LIN {X 0,Y 530.663,Z 618.387,A -85,B 0,C 180,E1 -4307.378,E2 -4307.378} C_VEL
LIN {X 0,Y 530.971,Z 618.347,A -85,B 0,C 180,E1 -4309.321,E2 -4309.321} C_VEL
LIN {X 0,Y 531.057,Z 618.337,A -85,B 0,C 180,E1 -4311.629,E2 -4311.629} C_VEL
LIN {X 0,Y 531.122,Z 618.328,A -85,B 0,C 180,E1 -4314.685,E2 -4314.685} C_VEL
LIN {X 0,Y 531.137,Z 618.326,A -85,B 0,C 180,E1 -4317.725,E2 -4317.725} C_VEL
LIN {X 0,Y 531.153,Z 618.324,A -85,B 0,C 180,E1 -4320.758,E2 -4320.758} C_VEL
LIN {X 0,Y 531.106,Z 618.33,A -85,B 0,C 180,E1 -4323.034,E2 -4323.034} C_VEL
LIN {X 0,Y 531.081,Z 618.333,A -85,B 0,C 180,E1 -4326.077,E2 -4326.077} C_VEL
LIN {X 0,Y 531.033,Z 618.339,A -85,B 0,C 180,E1 -4329.138,E2 -4329.138} C_VEL
LIN {X 0,Y 531.038,Z 618.338,A -85,B 0,C 180,E1 -4332.225,E2 -4332.225} C_VEL
LIN {X 0,Y 530.992,Z 618.344,A -85,B 0,C 180,E1 -4335.35,E2 -4335.35} C_VEL
LIN {X 0,Y 531.013,Z 618.343,A -85,B 0,C 180,E1 -4337.723,E2 -4337.723} C_VEL
LIN {X 0,Y 530.997,Z 618.345,A -85,B 0,C 180,E1 -4340.938,E2 -4340.938} C_VEL
LIN {X 0,Y 530.977,Z 618.346,A -85,B 0,C 180,E1 -4344.225,E2 -4344.225} C_VEL
LIN {X 0,Y 531.01,Z 618.342,A -85,B 0,C 180,E1 -4346.743,E2 -4346.743} C_VEL
LIN {X 0,Y 530.998,Z 618.344,A -85,B 0,C 180,E1 -4349.322,E2 -4349.322} C_VEL
LIN {X 0,Y 530.978,Z 618.348,A -85,B 0,C 180,E1 -4352.103,E2 -4352.103} C_VEL
LIN {X 0,Y 530.981,Z 618.345,A -85,B 0,C 180,E1 -4354.854,E2 -4354.854} C_VEL
LIN {X 0,Y 530.964,Z 618.348,A -85,B 0,C 180,E1 -4357.508,E2 -4357.508} C_VEL
LIN {X 0,Y 530.984,Z 618.347,A -85,B 0,C 180,E1 -4360.433,E2 -4360.433} C_VEL
LIN {X 0,Y 530.958,Z 618.349,A -85,B 0,C 180,E1 -4363.281,E2 -4363.281} C_VEL
LIN {X 0,Y 530.986,Z 618.347,A -85,B 0,C 180,E1 -4365.621,E2 -4365.621} C_VEL
LIN {X 0,Y 530.996,Z 618.346,A -85,B 0,C 180,E1 -4368.565,E2 -4368.565} C_VEL
LIN {X 0,Y 530.957,Z 618.35,A -85,B 0,C 180,E1 -4371.53,E2 -4371.53} C_VEL
LIN {X 0,Y 531.014,Z 618.346,A -85,B 0,C 180,E1 -4372.571,E2 -4372.571} C_VEL
LIN {X 0,Y 531.595,Z 622.566,A -85,B 0,C 180,E1 -4374.43,E2 -4374.43} C_VEL
LIN {X 0,Y 531.454,Z 629.172,A -85,B 0,C 180,E1 -4377.168,E2 -4377.168} C_VEL
LIN {X 0,Y 531.261,Z 636.953,A -85,B 0,C 180,E1 -4380.259,E2 -4380.259} C_VEL
LIN {X 0,Y 531.122,Z 644.77,A -85,B 0,C 180,E1 -4383.263,E2 -4383.263} C_VEL
LIN {X 0,Y 531.013,Z 651.98,A -85,B 0,C 180,E1 -4385.955,E2 -4385.955} C_VEL
LIN {X 0,Y 530.894,Z 659.398,A -85,B 0,C 180,E1 -4388.652,E2 -4388.652} C_VEL
LIN {X 0,Y 530.792,Z 667.357,A -85,B 0,C 180,E1 -4391.472,E2 -4391.472} C_VEL
LIN {X 0,Y 530.717,Z 676.275,A -85,B 0,C 180,E1 -4394.642,E2 -4394.642} C_VEL
LIN {X 0,Y 530.629,Z 681.493,A -85,B 0,C 180,E1 -4396.477,E2 -4396.477} C_VEL
LIN {X 0,Y 532.276,Z 692.282,A -85,B 0,C 180,E1 -4396.762,E2 -4396.762} C_VEL
LIN {X 0,Y 532.099,Z 704.784,A -85,B 0,C 180,E1 -4397.17,E2 -4397.17} C_VEL
LIN {X 0,Y 531.858,Z 716.415,A -85,B 0,C 180,E1 -4397.698,E2 -4397.698} C_VEL
LIN {X 0,Y 531.642,Z 727.398,A -85,B 0,C 180,E1 -4398.346,E2 -4398.346} C_VEL
LIN {X 0,Y 531.403,Z 738.098,A -85,B 0,C 180,E1 -4399.137,E2 -4399.137} C_VEL
LIN {X 0,Y 531.113,Z 748.543,A -85,B 0,C 180,E1 -4400.095,E2 -4400.095} C_VEL
LIN {X 0,Y 530.931,Z 756.994,A -85,B 0,C 180,E1 -4401.052,E2 -4401.052} C_VEL
LIN {X 0,Y 530.758,Z 765.238,A -85,B 0,C 180,E1 -4402.2,E2 -4402.2} C_VEL
LIN {X 0,Y 530.597,Z 772.271,A -85,B 0,C 180,E1 -4403.419,E2 -4403.419} C_VEL
LIN {X 0,Y 530.524,Z 777.951,A -85,B 0,C 180,E1 -4404.68,E2 -4404.68} C_VEL
LIN {X 0,Y 530.522,Z 781.896,A -85,B 0,C 180,E1 -4405.822,E2 -4405.822} C_VEL
LIN {X 0,Y 530.457,Z 784.808,A -85,B 0,C 180,E1 -4406.962,E2 -4406.962} C_VEL
LIN {X 0,Y 530.411,Z 786.195,A -85,B 0,C 180,E1 -4407.722,E2 -4407.722} C_VEL
LIN {X 0,Y 530.344,Z 787.786,A -85,B 0,C 180,E1 -4409.241,E2 -4409.241} C_VEL
LIN {X 0,Y 530.342,Z 788,A -85,B 0,C 180,E1 -4410,E2 -4410} C_VEL
LIN {X 0,Y 530.361,Z 787.184,A -85,B 0,C 180,E1 -4411.519,E2 -4411.519} C_VEL
LIN {X 0,Y 530.411,Z 786.197,A -85,B 0,C 180,E1 -4412.278,E2 -4412.278} C_VEL
LIN {X 0,Y 530.457,Z 784.809,A -85,B 0,C 180,E1 -4413.038,E2 -4413.038} C_VEL
LIN {X 0,Y 530.523,Z 781.895,A -85,B 0,C 180,E1 -4414.179,E2 -4414.179} C_VEL
LIN {X 0,Y 530.524,Z 777.947,A -85,B 0,C 180,E1 -4415.321,E2 -4415.321} C_VEL
LIN {X 0,Y 530.599,Z 772.261,A -85,B 0,C 180,E1 -4416.582,E2 -4416.582} C_VEL
LIN {X 0,Y 530.758,Z 765.234,A -85,B 0,C 180,E1 -4417.801,E2 -4417.801} C_VEL
LIN {X 0,Y 530.931,Z 756.989,A -85,B 0,C 180,E1 -4418.948,E2 -4418.948} C_VEL
LIN {X 0,Y 531.114,Z 748.537,A -85,B 0,C 180,E1 -4419.906,E2 -4419.906} C_VEL
LIN {X 0,Y 531.413,Z 738.09,A -85,B 0,C 180,E1 -4420.863,E2 -4420.863} C_VEL
LIN {X 0,Y 531.646,Z 727.379,A -85,B 0,C 180,E1 -4421.655,E2 -4421.655} C_VEL
LIN {X 0,Y 531.855,Z 716.401,A -85,B 0,C 180,E1 -4422.303,E2 -4422.303} C_VEL
LIN {X 0,Y 532.099,Z 704.757,A -85,B 0,C 180,E1 -4422.83,E2 -4422.83} C_VEL
LIN {X 0,Y 532.245,Z 691.335,A -85,B 0,C 180,E1 -4423.264,E2 -4423.264} C_VEL
LIN {X 0,Y 530.627,Z 681.491,A -85,B 0,C 180,E1 -4423.524,E2 -4423.524} C_VEL
LIN {X 0,Y 530.719,Z 674.047,A -85,B 0,C 180,E1 -4426.147,E2 -4426.147} C_VEL
LIN {X 0,Y 530.803,Z 666.211,A -85,B 0,C 180,E1 -4428.929,E2 -4428.929} C_VEL
LIN {X 0,Y 530.896,Z 659.342,A -85,B 0,C 180,E1 -4431.349,E2 -4431.349} C_VEL
LIN {X 0,Y 531.001,Z 651.365,A -85,B 0,C 180,E1 -4434.224,E2 -4434.224} C_VEL
LIN {X 0,Y 531.149,Z 643.534,A -85,B 0,C 180,E1 -4437.147,E2 -4437.147} C_VEL
LIN {X 0,Y 531.242,Z 635.619,A -85,B 0,C 180,E1 -4440.18,E2 -4440.18} C_VEL
LIN {X 0,Y 531.438,Z 628.98,A -85,B 0,C 180,E1 -4442.834,E2 -4442.834} C_VEL
LIN {X 0,Y 531.567,Z 622.445,A -85,B 0,C 180,E1 -4445.573,E2 -4445.573} C_VEL
LIN {X 0,Y 531.01,Z 618.343,A -85,B 0,C 180,E1 -4447.504,E2 -4447.504} C_VEL
LIN {X 0,Y 530.984,Z 618.348,A -85,B 0,C 180,E1 -4450.433,E2 -4450.433} C_VEL
LIN {X 0,Y 530.973,Z 618.349,A -85,B 0,C 180,E1 -4453.282,E2 -4453.282} C_VEL
LIN {X 0,Y 530.983,Z 618.346,A -85,B 0,C 180,E1 -4455.622,E2 -4455.622} C_VEL
LIN {X 0,Y 530.998,Z 618.345,A -85,B 0,C 180,E1 -4458.565,E2 -4458.565} C_VEL
LIN {X 0,Y 530.96,Z 618.35,A -85,B 0,C 180,E1 -4461.529,E2 -4461.529} C_VEL
LIN {X 0,Y 530.965,Z 618.349,A -85,B 0,C 180,E1 -4464.381,E2 -4464.381} C_VEL
LIN {X 0,Y 530.973,Z 618.347,A -85,B 0,C 180,E1 -4467.134,E2 -4467.134} C_VEL
LIN {X 0,Y 530.972,Z 618.347,A -85,B 0,C 180,E1 -4469.803,E2 -4469.803} C_VEL
LIN {X 0,Y 531.017,Z 618.343,A -85,B 0,C 180,E1 -4472.467,E2 -4472.467} C_VEL
LIN {X 0,Y 531.008,Z 618.342,A -85,B 0,C 180,E1 -4474.942,E2 -4474.942} C_VEL
LIN {X 0,Y 530.973,Z 618.347,A -85,B 0,C 180,E1 -4478.247,E2 -4478.247} C_VEL
LIN {X 0,Y 530.998,Z 618.345,A -85,B 0,C 180,E1 -4480.677,E2 -4480.677} C_VEL
LIN {X 0,Y 530.988,Z 618.345,A -85,B 0,C 180,E1 -4483.071,E2 -4483.071} C_VEL
LIN {X 0,Y 531.021,Z 618.342,A -85,B 0,C 180,E1 -4485.436,E2 -4485.436} C_VEL
LIN {X 0,Y 531.038,Z 618.34,A -85,B 0,C 180,E1 -4488.55,E2 -4488.55} C_VEL
LIN {X 0,Y 531.059,Z 618.338,A -85,B 0,C 180,E1 -4491.63,E2 -4491.63} C_VEL
LIN {X 0,Y 531.123,Z 618.33,A -85,B 0,C 180,E1 -4494.685,E2 -4494.685} C_VEL
LIN {X 0,Y 531.139,Z 618.328,A -85,B 0,C 180,E1 -4497.725,E2 -4497.725} C_VEL
LIN {X 0,Y 531.157,Z 618.326,A -85,B 0,C 180,E1 -4500.758,E2 -4500.758} C_VEL
LIN {X 0,Y 531.11,Z 618.331,A -85,B 0,C 180,E1 -4503.034,E2 -4503.034} C_VEL
LIN {X 0,Y 531.088,Z 618.333,A -85,B 0,C 180,E1 -4506.077,E2 -4506.077} C_VEL
LIN {X 0,Y 531.053,Z 618.338,A -85,B 0,C 180,E1 -4508.371,E2 -4508.371} C_VEL
LIN {X 0,Y 530.909,Z 618.469,A -85,B 0,C 180,E1 -4509.909,E2 -4509.909} C_VEL
LIN {X 0,Y 530.88,Z 621.989,A -85,B 0,C 180,E1 -4512.229,E2 -4512.229} C_VEL
LIN {X 0,Y 530.778,Z 626.84,A -85,B 0,C 180,E1 -4515.356,E2 -4515.356} C_VEL
LIN {X 0,Y 530.74,Z 630.57,A -85,B 0,C 180,E1 -4517.732,E2 -4517.732} C_VEL
LIN {X 0,Y 530.67,Z 635.636,A -85,B 0,C 180,E1 -4520.952,E2 -4520.952} C_VEL
LIN {X 0,Y 530.559,Z 640.479,A -85,B 0,C 180,E1 -4523.936,E2 -4523.936} C_VEL
LIN {X 0,Y 530.5,Z 645.195,A -85,B 0,C 180,E1 -4526.771,E2 -4526.771} C_VEL
LIN {X 0,Y 530.43,Z 649.68,A -85,B 0,C 180,E1 -4529.356,E2 -4529.356} C_VEL
LIN {X 0,Y 530.472,Z 653.555,A -85,B 0,C 180,E1 -4531.555,E2 -4531.555} C_VEL
LIN {X 0,Y 532.25,Z 665.028,A -85,B 0,C 180,E1 -4531.882,E2 -4531.882} C_VEL
LIN {X 0,Y 532.035,Z 677.886,A -85,B 0,C 180,E1 -4532.344,E2 -4532.344} C_VEL
LIN {X 0,Y 531.753,Z 689.78,A -85,B 0,C 180,E1 -4532.925,E2 -4532.925} C_VEL
LIN {X 0,Y 531.596,Z 700.528,A -85,B 0,C 180,E1 -4533.603,E2 -4533.603} C_VEL
LIN {X 0,Y 531.309,Z 711.099,A -85,B 0,C 180,E1 -4534.436,E2 -4534.436} C_VEL
LIN {X 0,Y 531.089,Z 721.098,A -85,B 0,C 180,E1 -4535.414,E2 -4535.414} C_VEL
LIN {X 0,Y 530.84,Z 730.038,A -85,B 0,C 180,E1 -4536.493,E2 -4536.493} C_VEL
LIN {X 0,Y 530.094,Z 733.676,A -85,B 0,C 180,E1 -4536.99,E2 -4536.99} C_VEL
LIN {X 0,Y 527.12,Z 739.135,A -85,B 0,C 180,E1 -4537.829,E2 -4537.829} C_VEL
LIN {X 0,Y 524.164,Z 743.924,A -85,B 0,C 180,E1 -4538.723,E2 -4538.723} C_VEL
LIN {X 0,Y 523.455,Z 746.507,A -85,B 0,C 180,E1 -4539.301,E2 -4539.301} C_VEL
LIN {X 0,Y 523.362,Z 751.369,A -85,B 0,C 180,E1 -4540.639,E2 -4540.639} C_VEL
LIN {X 0,Y 523.387,Z 754.149,A -85,B 0,C 180,E1 -4541.677,E2 -4541.677} C_VEL
LIN {X 0,Y 523.327,Z 755.607,A -85,B 0,C 180,E1 -4542.386,E2 -4542.386} C_VEL
LIN {X 0,Y 523.259,Z 757.186,A -85,B 0,C 180,E1 -4543.507,E2 -4543.507} C_VEL
LIN {X 0,Y 523.286,Z 757.918,A -85,B 0,C 180,E1 -4544.617,E2 -4544.617} C_VEL
LIN {X 0,Y 523.287,Z 757.853,A -85,B 0,C 180,E1 -4545.702,E2 -4545.702} C_VEL
LIN {X 0,Y 523.268,Z 756.994,A -85,B 0,C 180,E1 -4546.766,E2 -4546.766} C_VEL
LIN {X 0,Y 523.348,Z 755.384,A -85,B 0,C 180,E1 -4547.821,E2 -4547.821} C_VEL
LIN {X 0,Y 523.382,Z 753.069,A -85,B 0,C 180,E1 -4548.854,E2 -4548.854} C_VEL
LIN {X 0,Y 523.421,Z 749.79,A -85,B 0,C 180,E1 -4549.938,E2 -4549.938} C_VEL
LIN {X 0,Y 523.475,Z 745.006,A -85,B 0,C 180,E1 -4551.141,E2 -4551.141} C_VEL
LIN {X 0,Y 523.592,Z 738.759,A -85,B 0,C 180,E1 -4552.367,E2 -4552.367} C_VEL
LIN {X 0,Y 523.795,Z 730.757,A -85,B 0,C 180,E1 -4553.615,E2 -4553.615} C_VEL
LIN {X 0,Y 524.056,Z 721.306,A -85,B 0,C 180,E1 -4554.784,E2 -4554.784} C_VEL
LIN {X 0,Y 524.295,Z 711.765,A -85,B 0,C 180,E1 -4555.737,E2 -4555.737} C_VEL
LIN {X 0,Y 524.573,Z 701.221,A -85,B 0,C 180,E1 -4556.592,E2 -4556.592} C_VEL
LIN {X 0,Y 524.864,Z 689.192,A -85,B 0,C 180,E1 -4557.359,E2 -4557.359} C_VEL
LIN {X 0,Y 525.157,Z 676.521,A -85,B 0,C 180,E1 -4557.975,E2 -4557.975} C_VEL
LIN {X 0,Y 525.253,Z 664.446,A -85,B 0,C 180,E1 -4558.404,E2 -4558.404} C_VEL
LIN {X 0,Y 523.387,Z 653.54,A -85,B 0,C 180,E1 -4558.729,E2 -4558.729} C_VEL
LIN {X 0,Y 523.403,Z 648.016,A -85,B 0,C 180,E1 -4561.968,E2 -4561.968} C_VEL
LIN {X 0,Y 523.421,Z 643.715,A -85,B 0,C 180,E1 -4564.553,E2 -4564.553} C_VEL
LIN {X 0,Y 523.504,Z 639.577,A -85,B 0,C 180,E1 -4567.087,E2 -4567.087} C_VEL
LIN {X 0,Y 523.62,Z 634.259,A -85,B 0,C 180,E1 -4570.394,E2 -4570.394} C_VEL
LIN {X 0,Y 523.691,Z 630.378,A -85,B 0,C 180,E1 -4572.828,E2 -4572.828} C_VEL
LIN {X 0,Y 523.776,Z 626.626,A -85,B 0,C 180,E1 -4575.23,E2 -4575.23} C_VEL
LIN {X 0,Y 523.893,Z 621.736,A -85,B 0,C 180,E1 -4578.391,E2 -4578.391} C_VEL
LIN {X 0,Y 523.823,Z 619.373,A -85,B 0,C 180,E1 -4579.955,E2 -4579.955} C_VEL
LIN {X 0,Y 524.032,Z 619.21,A -85,B 0,C 180,E1 -4582.292,E2 -4582.292} C_VEL
LIN {X 0,Y 524.084,Z 619.205,A -85,B 0,C 180,E1 -4584.613,E2 -4584.613} C_VEL
LIN {X 0,Y 524.117,Z 619.199,A -85,B 0,C 180,E1 -4587.694,E2 -4587.694} C_VEL
LIN {X 0,Y 524.128,Z 619.201,A -85,B 0,C 180,E1 -4590.768,E2 -4590.768} C_VEL
LIN {X 0,Y 524.075,Z 619.208,A -85,B 0,C 180,E1 -4593.075,E2 -4593.075} C_VEL
LIN {X 0,Y 524.046,Z 619.208,A -85,B 0,C 180,E1 -4596.159,E2 -4596.159} C_VEL
LIN {X 0,Y 523.95,Z 619.221,A -85,B 0,C 180,E1 -4598.485,E2 -4598.485} C_VEL
LIN {X 0,Y 523.674,Z 619.358,A -85,B 0,C 180,E1 -4600.536,E2 -4600.536} C_VEL
LIN {X 0,Y 523.624,Z 624.031,A -85,B 0,C 180,E1 -4603.189,E2 -4603.189} C_VEL
LIN {X 0,Y 523.625,Z 628.196,A -85,B 0,C 180,E1 -4605.571,E2 -4605.571} C_VEL
LIN {X 0,Y 523.558,Z 632.361,A -85,B 0,C 180,E1 -4607.983,E2 -4607.983} C_VEL
LIN {X 0,Y 523.496,Z 636.576,A -85,B 0,C 180,E1 -4610.429,E2 -4610.429} C_VEL
LIN {X 0,Y 523.445,Z 640.835,A -85,B 0,C 180,E1 -4612.915,E2 -4612.915} C_VEL
LIN {X 0,Y 523.405,Z 645.914,A -85,B 0,C 180,E1 -4615.889,E2 -4615.889} C_VEL
LIN {X 0,Y 523.372,Z 651.027,A -85,B 0,C 180,E1 -4618.908,E2 -4618.908} C_VEL
LIN {X 0,Y 523.36,Z 653.567,A -85,B 0,C 180,E1 -4620.375,E2 -4620.375} C_VEL
LIN {X 0,Y 525.317,Z 665.093,A -85,B 0,C 180,E1 -4620.716,E2 -4620.716} C_VEL
LIN {X 0,Y 525.15,Z 675.335,A -85,B 0,C 180,E1 -4621.074,E2 -4621.074} C_VEL
LIN {X 0,Y 524.93,Z 685.377,A -85,B 0,C 180,E1 -4621.532,E2 -4621.532} C_VEL
LIN {X 0,Y 524.657,Z 696.427,A -85,B 0,C 180,E1 -4622.172,E2 -4622.172} C_VEL
LIN {X 0,Y 524.356,Z 708.631,A -85,B 0,C 180,E1 -4623.082,E2 -4623.082} C_VEL
LIN {X 0,Y 524.136,Z 716.799,A -85,B 0,C 180,E1 -4623.833,E2 -4623.833} C_VEL
LIN {X 0,Y 523.903,Z 725.166,A -85,B 0,C 180,E1 -4624.758,E2 -4624.758} C_VEL
LIN {X 0,Y 523.744,Z 732.355,A -85,B 0,C 180,E1 -4625.712,E2 -4625.712} C_VEL
LIN {X 0,Y 523.585,Z 738.747,A -85,B 0,C 180,E1 -4626.731,E2 -4626.731} C_VEL
LIN {X 0,Y 523.506,Z 743.425,A -85,B 0,C 180,E1 -4627.621,E2 -4627.621} C_VEL
LIN {X 0,Y 523.423,Z 748.629,A -85,B 0,C 180,E1 -4628.852,E2 -4628.852} C_VEL
LIN {X 0,Y 523.314,Z 752.5,A -85,B 0,C 180,E1 -4630.048,E2 -4630.048} C_VEL
LIN {X 0,Y 523.276,Z 755.254,A -85,B 0,C 180,E1 -4631.225,E2 -4631.225} C_VEL
LIN {X 0,Y 523.28,Z 757.001,A -85,B 0,C 180,E1 -4632.38,E2 -4632.38} C_VEL
LIN {X 0,Y 523.242,Z 757.828,A -85,B 0,C 180,E1 -4633.505,E2 -4633.505} C_VEL
LIN {X 0,Y 523.282,Z 757.815,A -85,B 0,C 180,E1 -4634.616,E2 -4634.616} C_VEL
LIN {X 0,Y 523.283,Z 757.01,A -85,B 0,C 180,E1 -4635.702,E2 -4635.702} C_VEL
LIN {X 0,Y 523.27,Z 755.448,A -85,B 0,C 180,E1 -4636.766,E2 -4636.766} C_VEL
LIN {X 0,Y 523.369,Z 753.109,A -85,B 0,C 180,E1 -4637.823,E2 -4637.823} C_VEL
LIN {X 0,Y 523.413,Z 750.022,A -85,B 0,C 180,E1 -4638.857,E2 -4638.857} C_VEL
LIN {X 0,Y 523.471,Z 745.899,A -85,B 0,C 180,E1 -4639.93,E2 -4639.93} C_VEL
LIN {X 0,Y 523.602,Z 740.066,A -85,B 0,C 180,E1 -4641.122,E2 -4641.122} C_VEL
LIN {X 0,Y 523.695,Z 733.955,A -85,B 0,C 180,E1 -4642.14,E2 -4642.14} C_VEL
LIN {X 0,Y 523.839,Z 727.364,A -85,B 0,C 180,E1 -4643.056,E2 -4643.056} C_VEL
LIN {X 0,Y 524.024,Z 720.787,A -85,B 0,C 180,E1 -4643.835,E2 -4643.835} C_VEL
LIN {X 0,Y 524.293,Z 712.256,A -85,B 0,C 180,E1 -4644.684,E2 -4644.684} C_VEL
LIN {X 0,Y 524.466,Z 703.684,A -85,B 0,C 180,E1 -4645.4,E2 -4645.4} C_VEL
LIN {X 0,Y 524.715,Z 695.335,A -85,B 0,C 180,E1 -4645.985,E2 -4645.985} C_VEL
LIN {X 0,Y 524.938,Z 685.305,A -85,B 0,C 180,E1 -4646.561,E2 -4646.561} C_VEL
LIN {X 0,Y 525.181,Z 675.463,A -85,B 0,C 180,E1 -4647.011,E2 -4647.011} C_VEL
LIN {X 0,Y 525.36,Z 665.364,A -85,B 0,C 180,E1 -4647.365,E2 -4647.365} C_VEL
LIN {X 0,Y 523.477,Z 654.705,A -85,B 0,C 180,E1 -4647.684,E2 -4647.684} C_VEL
LIN {X 0,Y 523.353,Z 653.563,A -85,B 0,C 180,E1 -4647.717,E2 -4647.717} C_VEL
LIN {X 0,Y 523.413,Z 647.795,A -85,B 0,C 180,E1 -4651.093,E2 -4651.093} C_VEL
LIN {X 0,Y 523.469,Z 642.776,A -85,B 0,C 180,E1 -4654.095,E2 -4654.095} C_VEL
LIN {X 0,Y 523.494,Z 637.504,A -85,B 0,C 180,E1 -4657.087,E2 -4657.087} C_VEL
LIN {X 0,Y 523.523,Z 632.382,A -85,B 0,C 180,E1 -4660.001,E2 -4660.001} C_VEL
LIN {X 0,Y 523.573,Z 627.302,A -85,B 0,C 180,E1 -4662.824,E2 -4662.824} C_VEL
LIN {X 0,Y 523.651,Z 622.868,A -85,B 0,C 180,E1 -4665.226,E2 -4665.226} C_VEL
LIN {X 0,Y 523.584,Z 619.269,A -85,B 0,C 180,E1 -4667.204,E2 -4667.204} C_VEL
LIN {X 0,Y 523.91,Z 619.228,A -85,B 0,C 180,E1 -4669.175,E2 -4669.175} C_VEL
LIN {X 0,Y 524.005,Z 619.215,A -85,B 0,C 180,E1 -4671.516,E2 -4671.516} C_VEL
LIN {X 0,Y 524.083,Z 619.205,A -85,B 0,C 180,E1 -4674.614,E2 -4674.614} C_VEL
LIN {X 0,Y 524.109,Z 619.201,A -85,B 0,C 180,E1 -4677.694,E2 -4677.694} C_VEL
LIN {X 0,Y 524.122,Z 619.2,A -85,B 0,C 180,E1 -4680.768,E2 -4680.768} C_VEL
LIN {X 0,Y 524.073,Z 619.207,A -85,B 0,C 180,E1 -4683.075,E2 -4683.075} C_VEL
LIN {X 0,Y 524.043,Z 619.21,A -85,B 0,C 180,E1 -4686.159,E2 -4686.159} C_VEL
LIN {X 0,Y 524.001,Z 619.215,A -85,B 0,C 180,E1 -4689.262,E2 -4689.262} C_VEL
LIN {X 0,Y 524.005,Z 619.215,A -85,B 0,C 180,E1 -4691.743,E2 -4691.743} C_VEL
LIN {X 0,Y 523.989,Z 619.217,A -85,B 0,C 180,E1 -4695.053,E2 -4695.053} C_VEL
LIN {X 0,Y 523.961,Z 619.221,A -85,B 0,C 180,E1 -4697.969,E2 -4697.969} C_VEL
LIN {X 0,Y 523.968,Z 619.219,A -85,B 0,C 180,E1 -4700.41,E2 -4700.41} C_VEL
LIN {X 0,Y 523.914,Z 619.228,A -85,B 0,C 180,E1 -4702.893,E2 -4702.893} C_VEL
LIN {X 0,Y 523.952,Z 619.221,A -85,B 0,C 180,E1 -4705.419,E2 -4705.419} C_VEL
LIN {X 0,Y 523.968,Z 619.221,A -85,B 0,C 180,E1 -4707.999,E2 -4707.999} C_VEL
LIN {X 0,Y 523.95,Z 619.221,A -85,B 0,C 180,E1 -4710.857,E2 -4710.857} C_VEL
LIN {X 0,Y 523.958,Z 619.22,A -85,B 0,C 180,E1 -4713.735,E2 -4713.735} C_VEL
LIN {X 0,Y 523.917,Z 619.227,A -85,B 0,C 180,E1 -4716.404,E2 -4716.404} C_VEL
LIN {X 0,Y 523.921,Z 619.225,A -85,B 0,C 180,E1 -4719.085,E2 -4719.085} C_VEL
LIN {X 0,Y 523.951,Z 619.221,A -85,B 0,C 180,E1 -4722.119,E2 -4722.119} C_VEL
LIN {X 0,Y 523.954,Z 619.222,A -85,B 0,C 180,E1 -4725.309,E2 -4725.309} C_VEL
LIN {X 0,Y 523.958,Z 619.223,A -85,B 0,C 180,E1 -4728.69,E2 -4728.69} C_VEL
LIN {X 0,Y 523.928,Z 619.226,A -85,B 0,C 180,E1 -4731.9,E2 -4731.9} C_VEL
LIN {X 0,Y 524,Z 619.385,A -85,B 0,C 180,E1 -4732.461,E2 -4732.461} C_VEL
LIN {X 0,Y 524.592,Z 623.625,A -85,B 0,C 180,E1 -4734.355,E2 -4734.355} C_VEL
LIN {X 0,Y 524.469,Z 630.231,A -85,B 0,C 180,E1 -4737.132,E2 -4737.132} C_VEL
LIN {X 0,Y 524.245,Z 638.005,A -85,B 0,C 180,E1 -4740.264,E2 -4740.264} C_VEL
LIN {X 0,Y 524.09,Z 645.801,A -85,B 0,C 180,E1 -4743.306,E2 -4743.306} C_VEL
LIN {X 0,Y 523.933,Z 653.646,A -85,B 0,C 180,E1 -4746.271,E2 -4746.271} C_VEL
LIN {X 0,Y 523.821,Z 661.531,A -85,B 0,C 180,E1 -4749.174,E2 -4749.174} C_VEL
LIN {X 0,Y 523.707,Z 669.486,A -85,B 0,C 180,E1 -4752.022,E2 -4752.022} C_VEL
LIN {X 0,Y 523.617,Z 678.502,A -85,B 0,C 180,E1 -4755.226,E2 -4755.226} C_VEL
LIN {X 0,Y 523.573,Z 681.493,A -85,B 0,C 180,E1 -4756.291,E2 -4756.291} C_VEL
LIN {X 0,Y 525.365,Z 693.197,A -85,B 0,C 180,E1 -4756.609,E2 -4756.609} C_VEL
LIN {X 0,Y 525.168,Z 705.99,A -85,B 0,C 180,E1 -4757.047,E2 -4757.047} C_VEL
LIN {X 0,Y 524.891,Z 718.179,A -85,B 0,C 180,E1 -4757.63,E2 -4757.63} C_VEL
LIN {X 0,Y 524.677,Z 729.211,A -85,B 0,C 180,E1 -4758.314,E2 -4758.314} C_VEL
LIN {X 0,Y 524.362,Z 740.403,A -85,B 0,C 180,E1 -4759.185,E2 -4759.185} C_VEL
LIN {X 0,Y 524.086,Z 750.336,A -85,B 0,C 180,E1 -4760.156,E2 -4760.156} C_VEL
LIN {X 0,Y 523.851,Z 759.963,A -85,B 0,C 180,E1 -4761.32,E2 -4761.32} C_VEL
LIN {X 0,Y 523.633,Z 767.624,A -85,B 0,C 180,E1 -4762.481,E2 -4762.481} C_VEL
LIN {X 0,Y 523.515,Z 774.681,A -85,B 0,C 180,E1 -4763.835,E2 -4763.835} C_VEL
LIN {X 0,Y 523.383,Z 779.374,A -85,B 0,C 180,E1 -4764.993,E2 -4764.993} C_VEL
LIN {X 0,Y 523.443,Z 782.959,A -85,B 0,C 180,E1 -4766.151,E2 -4766.151} C_VEL
LIN {X 0,Y 523.367,Z 784.808,A -85,B 0,C 180,E1 -4766.921,E2 -4766.921} C_VEL
LIN {X 0,Y 523.334,Z 786.195,A -85,B 0,C 180,E1 -4767.691,E2 -4767.691} C_VEL
LIN {X 0,Y 523.25,Z 787.786,A -85,B 0,C 180,E1 -4769.231,E2 -4769.231} C_VEL
LIN {X 0,Y 523.246,Z 788,A -85,B 0,C 180,E1 -4770,E2 -4770} C_VEL
LIN {X 0,Y 523.274,Z 787.184,A -85,B 0,C 180,E1 -4771.54,E2 -4771.54} C_VEL
LIN {X 0,Y 523.335,Z 786.196,A -85,B 0,C 180,E1 -4772.309,E2 -4772.309} C_VEL
LIN {X 0,Y 523.367,Z 784.809,A -85,B 0,C 180,E1 -4773.079,E2 -4773.079} C_VEL
LIN {X 0,Y 523.442,Z 781.894,A -85,B 0,C 180,E1 -4774.235,E2 -4774.235} C_VEL
LIN {X 0,Y 523.464,Z 777.947,A -85,B 0,C 180,E1 -4775.393,E2 -4775.393} C_VEL
LIN {X 0,Y 523.524,Z 772.725,A -85,B 0,C 180,E1 -4776.581,E2 -4776.581} C_VEL
LIN {X 0,Y 523.665,Z 766.465,A -85,B 0,C 180,E1 -4777.713,E2 -4777.713} C_VEL
LIN {X 0,Y 523.857,Z 758.475,A -85,B 0,C 180,E1 -4778.875,E2 -4778.875} C_VEL
LIN {X 0,Y 524.086,Z 750.331,A -85,B 0,C 180,E1 -4779.845,E2 -4779.845} C_VEL
LIN {X 0,Y 524.37,Z 740.394,A -85,B 0,C 180,E1 -4780.815,E2 -4780.815} C_VEL
LIN {X 0,Y 524.64,Z 729.192,A -85,B 0,C 180,E1 -4781.688,E2 -4781.688} C_VEL
LIN {X 0,Y 524.845,Z 718.167,A -85,B 0,C 180,E1 -4782.372,E2 -4782.372} C_VEL
LIN {X 0,Y 525.147,Z 705.966,A -85,B 0,C 180,E1 -4782.954,E2 -4782.954} C_VEL
LIN {X 0,Y 525.365,Z 693.164,A -85,B 0,C 180,E1 -4783.391,E2 -4783.391} C_VEL
LIN {X 0,Y 523.57,Z 681.491,A -85,B 0,C 180,E1 -4783.71,E2 -4783.71} C_VEL
LIN {X 0,Y 523.648,Z 674.01,A -85,B 0,C 180,E1 -4786.371,E2 -4786.371} C_VEL
LIN {X 0,Y 523.757,Z 666.025,A -85,B 0,C 180,E1 -4789.193,E2 -4789.193} C_VEL
LIN {X 0,Y 523.855,Z 658.006,A -85,B 0,C 180,E1 -4792.064,E2 -4792.064} C_VEL
LIN {X 0,Y 523.977,Z 650.101,A -85,B 0,C 180,E1 -4794.993,E2 -4794.993} C_VEL
LIN {X 0,Y 524.123,Z 642.851,A -85,B 0,C 180,E1 -4797.748,E2 -4797.748} C_VEL
LIN {X 0,Y 524.256,Z 635.529,A -85,B 0,C 180,E1 -4800.625,E2 -4800.625} C_VEL
LIN {X 0,Y 524.451,Z 628.91,A -85,B 0,C 180,E1 -4803.328,E2 -4803.328} C_VEL
LIN {X 0,Y 524.567,Z 623.508,A -85,B 0,C 180,E1 -4805.647,E2 -4805.647} C_VEL
LIN {X 0,Y 523.944,Z 619.221,A -85,B 0,C 180,E1 -4807.683,E2 -4807.683} C_VEL
LIN {X 0,Y 523.94,Z 619.225,A -85,B 0,C 180,E1 -4810.13,E2 -4810.13} C_VEL
LIN {X 0,Y 523.942,Z 619.224,A -85,B 0,C 180,E1 -4812.459,E2 -4812.459} C_VEL
LIN {X 0,Y 523.953,Z 619.223,A -85,B 0,C 180,E1 -4815.309,E2 -4815.309} C_VEL
LIN {X 0,Y 523.96,Z 619.221,A -85,B 0,C 180,E1 -4818.689,E2 -4818.689} C_VEL
LIN {X 0,Y 523.92,Z 619.227,A -85,B 0,C 180,E1 -4821.08,E2 -4821.08} C_VEL
LIN {X 0,Y 523.908,Z 619.227,A -85,B 0,C 180,E1 -4823.826,E2 -4823.826} C_VEL
LIN {X 0,Y 523.944,Z 619.223,A -85,B 0,C 180,E1 -4826.636,E2 -4826.636} C_VEL
LIN {X 0,Y 523.958,Z 619.222,A -85,B 0,C 180,E1 -4829.356,E2 -4829.356} C_VEL
LIN {X 0,Y 523.98,Z 619.218,A -85,B 0,C 180,E1 -4832.281,E2 -4832.281} C_VEL
LIN {X 0,Y 523.955,Z 619.223,A -85,B 0,C 180,E1 -4834.581,E2 -4834.581} C_VEL
LIN {X 0,Y 523.917,Z 619.226,A -85,B 0,C 180,E1 -4837.107,E2 -4837.107} C_VEL
LIN {X 0,Y 523.981,Z 619.218,A -85,B 0,C 180,E1 -4839.866,E2 -4839.866} C_VEL
LIN {X 0,Y 523.969,Z 619.22,A -85,B 0,C 180,E1 -4842.837,E2 -4842.837} C_VEL
LIN {X 0,Y 523.979,Z 619.218,A -85,B 0,C 180,E1 -4845.236,E2 -4845.236} C_VEL
LIN {X 0,Y 524.014,Z 619.214,A -85,B 0,C 180,E1 -4848.394,E2 -4848.394} C_VEL
LIN {X 0,Y 524.007,Z 619.216,A -85,B 0,C 180,E1 -4851.516,E2 -4851.516} C_VEL
LIN {X 0,Y 524.085,Z 619.206,A -85,B 0,C 180,E1 -4854.614,E2 -4854.614} C_VEL
LIN {X 0,Y 524.112,Z 619.203,A -85,B 0,C 180,E1 -4857.694,E2 -4857.694} C_VEL
LIN {X 0,Y 524.127,Z 619.202,A -85,B 0,C 180,E1 -4860.768,E2 -4860.768} C_VEL
LIN {X 0,Y 524.076,Z 619.207,A -85,B 0,C 180,E1 -4863.075,E2 -4863.075} C_VEL
LIN {X 0,Y 524.05,Z 619.21,A -85,B 0,C 180,E1 -4866.159,E2 -4866.159} C_VEL
LIN {X 0,Y 523.998,Z 619.216,A -85,B 0,C 180,E1 -4868.484,E2 -4868.484} C_VEL
LIN {X 0,Y 523.871,Z 619.579,A -85,B 0,C 180,E1 -4870.044,E2 -4870.044} C_VEL
LIN {X 0,Y 523.845,Z 623.107,A -85,B 0,C 180,E1 -4872.396,E2 -4872.396} C_VEL
LIN {X 0,Y 523.725,Z 627.971,A -85,B 0,C 180,E1 -4875.568,E2 -4875.568} C_VEL
LIN {X 0,Y 523.675,Z 631.739,A -85,B 0,C 180,E1 -4877.979,E2 -4877.979} C_VEL
LIN {X 0,Y 523.601,Z 635.499,A -85,B 0,C 180,E1 -4880.425,E2 -4880.425} C_VEL
LIN {X 0,Y 523.511,Z 640.803,A -85,B 0,C 180,E1 -4883.75,E2 -4883.75} C_VEL
LIN {X 0,Y 523.437,Z 644.979,A -85,B 0,C 180,E1 -4886.301,E2 -4886.301} C_VEL
LIN {X 0,Y 523.376,Z 649.842,A -85,B 0,C 180,E1 -4889.21,E2 -4889.21} C_VEL
LIN {X 0,Y 523.383,Z 653.531,A -85,B 0,C 180,E1 -4891.355,E2 -4891.355} C_VEL
LIN {X 0,Y 525.332,Z 666.248,A -85,B 0,C 180,E1 -4891.745,E2 -4891.745} C_VEL
LIN {X 0,Y 525.101,Z 678.466,A -85,B 0,C 180,E1 -4892.199,E2 -4892.199} C_VEL
LIN {X 0,Y 524.815,Z 689.704,A -85,B 0,C 180,E1 -4892.758,E2 -4892.758} C_VEL
LIN {X 0,Y 524.607,Z 701.194,A -85,B 0,C 180,E1 -4893.497,E2 -4893.497} C_VEL
LIN {X 0,Y 524.277,Z 712.07,A -85,B 0,C 180,E1 -4894.381,E2 -4894.381} C_VEL
LIN {X 0,Y 524.042,Z 721.572,A -85,B 0,C 180,E1 -4895.335,E2 -4895.335} C_VEL
LIN {X 0,Y 523.792,Z 730.449,A -85,B 0,C 180,E1 -4896.432,E2 -4896.432} C_VEL
LIN {X 0,Y 523.592,Z 738.243,A -85,B 0,C 180,E1 -4897.633,E2 -4897.633} C_VEL
LIN {X 0,Y 523.479,Z 744.587,A -85,B 0,C 180,E1 -4898.86,E2 -4898.86} C_VEL
LIN {X 0,Y 523.455,Z 746.507,A -85,B 0,C 180,E1 -4899.301,E2 -4899.301} C_VEL
LIN {X 0,Y 522.754,Z 748.868,A -85,B 0,C 180,E1 -4899.89,E2 -4899.89} C_VEL
LIN {X 0,Y 519.837,Z 752.139,A -85,B 0,C 180,E1 -4900.869,E2 -4900.869} C_VEL
LIN {X 0,Y 517.38,Z 754.235,A -85,B 0,C 180,E1 -4901.676,E2 -4901.676} C_VEL
LIN {X 0,Y 516.313,Z 755.527,A -85,B 0,C 180,E1 -4902.307,E2 -4902.307} C_VEL
LIN {X 0,Y 516.219,Z 755.872,A -85,B 0,C 180,E1 -4902.521,E2 -4902.521} C_VEL
LIN {X 0,Y 516.187,Z 757.61,A -85,B 0,C 180,E1 -4903.978,E2 -4903.978} C_VEL
LIN {X 0,Y 516.194,Z 757.999,A -85,B 0,C 180,E1 -4905.071,E2 -4905.071} C_VEL
LIN {X 0,Y 516.181,Z 757.562,A -85,B 0,C 180,E1 -4906.188,E2 -4906.188} C_VEL
LIN {X 0,Y 516.204,Z 756.282,A -85,B 0,C 180,E1 -4907.324,E2 -4907.324} C_VEL
LIN {X 0,Y 516.267,Z 754.098,A -85,B 0,C 180,E1 -4908.48,E2 -4908.48} C_VEL
LIN {X 0,Y 516.297,Z 750.876,A -85,B 0,C 180,E1 -4909.667,E2 -4909.667} C_VEL
LIN {X 0,Y 516.383,Z 746.482,A -85,B 0,C 180,E1 -4910.875,E2 -4910.875} C_VEL
LIN {X 0,Y 516.528,Z 740.01,A -85,B 0,C 180,E1 -4912.245,E2 -4912.245} C_VEL
LIN {X 0,Y 516.704,Z 732.016,A -85,B 0,C 180,E1 -4913.55,E2 -4913.55} C_VEL
LIN {X 0,Y 516.959,Z 723.582,A -85,B 0,C 180,E1 -4914.656,E2 -4914.656} C_VEL
LIN {X 0,Y 517.193,Z 714.658,A -85,B 0,C 180,E1 -4915.614,E2 -4915.614} C_VEL
LIN {X 0,Y 517.534,Z 704.259,A -85,B 0,C 180,E1 -4916.518,E2 -4916.518} C_VEL
LIN {X 0,Y 517.854,Z 691.871,A -85,B 0,C 180,E1 -4917.372,E2 -4917.372} C_VEL
LIN {X 0,Y 518.117,Z 679.95,A -85,B 0,C 180,E1 -4918.004,E2 -4918.004} C_VEL
LIN {X 0,Y 518.413,Z 666.799,A -85,B 0,C 180,E1 -4918.509,E2 -4918.509} C_VEL
LIN {X 0,Y 516.547,Z 655.269,A -85,B 0,C 180,E1 -4918.867,E2 -4918.867} C_VEL
LIN {X 0,Y 516.285,Z 653.641,A -85,B 0,C 180,E1 -4918.915,E2 -4918.915} C_VEL
LIN {X 0,Y 516.337,Z 648.114,A -85,B 0,C 180,E1 -4922.219,E2 -4922.219} C_VEL
LIN {X 0,Y 516.348,Z 643.508,A -85,B 0,C 180,E1 -4925.043,E2 -4925.043} C_VEL
LIN {X 0,Y 516.429,Z 639.214,A -85,B 0,C 180,E1 -4927.729,E2 -4927.729} C_VEL
LIN {X 0,Y 516.543,Z 635.403,A -85,B 0,C 180,E1 -4930.114,E2 -4930.114} C_VEL
LIN {X 0,Y 516.615,Z 631.495,A -85,B 0,C 180,E1 -4932.585,E2 -4932.585} C_VEL
LIN {X 0,Y 516.713,Z 626.469,A -85,B 0,C 180,E1 -4935.828,E2 -4935.828} C_VEL
LIN {X 0,Y 516.845,Z 621.605,A -85,B 0,C 180,E1 -4939.025,E2 -4939.025} C_VEL
LIN {X 0,Y 516.778,Z 620.432,A -85,B 0,C 180,E1 -4939.817,E2 -4939.817} C_VEL
LIN {X 0,Y 516.953,Z 620.093,A -85,B 0,C 180,E1 -4941.399,E2 -4941.399} C_VEL
LIN {X 0,Y 517.013,Z 620.085,A -85,B 0,C 180,E1 -4943.757,E2 -4943.757} C_VEL
LIN {X 0,Y 517.089,Z 620.074,A -85,B 0,C 180,E1 -4947.663,E2 -4947.663} C_VEL
LIN {X 0,Y 517.098,Z 620.077,A -85,B 0,C 180,E1 -4950.778,E2 -4950.778} C_VEL
LIN {X 0,Y 517.016,Z 620.087,A -85,B 0,C 180,E1 -4953.117,E2 -4953.117} C_VEL
LIN {X 0,Y 517.01,Z 620.084,A -85,B 0,C 180,E1 -4956.243,E2 -4956.243} C_VEL
LIN {X 0,Y 516.914,Z 620.097,A -85,B 0,C 180,E1 -4958.601,E2 -4958.601} C_VEL
LIN {X 0,Y 516.628,Z 620.285,A -85,B 0,C 180,E1 -4960.681,E2 -4960.681} C_VEL
LIN {X 0,Y 516.561,Z 624.998,A -85,B 0,C 180,E1 -4963.373,E2 -4963.373} C_VEL
LIN {X 0,Y 516.539,Z 629.187,A -85,B 0,C 180,E1 -4965.79,E2 -4965.79} C_VEL
LIN {X 0,Y 516.478,Z 633.393,A -85,B 0,C 180,E1 -4968.238,E2 -4968.238} C_VEL
LIN {X 0,Y 516.406,Z 637.622,A -85,B 0,C 180,E1 -4970.722,E2 -4970.722} C_VEL
LIN {X 0,Y 516.364,Z 641.922,A -85,B 0,C 180,E1 -4973.247,E2 -4973.247} C_VEL
LIN {X 0,Y 516.323,Z 646.699,A -85,B 0,C 180,E1 -4976.055,E2 -4976.055} C_VEL
LIN {X 0,Y 516.272,Z 650.704,A -85,B 0,C 180,E1 -4978.454,E2 -4978.454} C_VEL
LIN {X 0,Y 516.279,Z 653.62,A -85,B 0,C 180,E1 -4980.181,E2 -4980.181} C_VEL
LIN {X 0,Y 518.377,Z 665.91,A -85,B 0,C 180,E1 -4980.558,E2 -4980.558} C_VEL
LIN {X 0,Y 518.183,Z 678.5,A -85,B 0,C 180,E1 -4981.023,E2 -4981.023} C_VEL
LIN {X 0,Y 517.856,Z 691.103,A -85,B 0,C 180,E1 -4981.677,E2 -4981.677} C_VEL
LIN {X 0,Y 517.562,Z 700.61,A -85,B 0,C 180,E1 -4982.302,E2 -4982.302} C_VEL
LIN {X 0,Y 517.339,Z 709.715,A -85,B 0,C 180,E1 -4983.03,E2 -4983.03} C_VEL
LIN {X 0,Y 517.107,Z 717.291,A -85,B 0,C 180,E1 -4983.747,E2 -4983.747} C_VEL
LIN {X 0,Y 516.874,Z 724.927,A -85,B 0,C 180,E1 -4984.601,E2 -4984.601} C_VEL
LIN {X 0,Y 516.684,Z 731.844,A -85,B 0,C 180,E1 -4985.521,E2 -4985.521} C_VEL
LIN {X 0,Y 516.554,Z 737.48,A -85,B 0,C 180,E1 -4986.402,E2 -4986.402} C_VEL
LIN {X 0,Y 516.453,Z 743.337,A -85,B 0,C 180,E1 -4987.514,E2 -4987.514} C_VEL
LIN {X 0,Y 516.38,Z 746.807,A -85,B 0,C 180,E1 -4988.287,E2 -4988.287} C_VEL
LIN {X 0,Y 516.288,Z 750.888,A -85,B 0,C 180,E1 -4989.419,E2 -4989.419} C_VEL
LIN {X 0,Y 516.199,Z 754.511,A -85,B 0,C 180,E1 -4990.806,E2 -4990.806} C_VEL
LIN {X 0,Y 516.187,Z 756.405,A -85,B 0,C 180,E1 -4991.846,E2 -4991.846} C_VEL
LIN {X 0,Y 516.168,Z 757.576,A -85,B 0,C 180,E1 -4992.904,E2 -4992.904} C_VEL
LIN {X 0,Y 516.179,Z 757.993,A -85,B 0,C 180,E1 -4993.978,E2 -4993.978} C_VEL
LIN {X 0,Y 516.19,Z 757.639,A -85,B 0,C 180,E1 -4995.071,E2 -4995.071} C_VEL
LIN {X 0,Y 516.18,Z 756.471,A -85,B 0,C 180,E1 -4996.187,E2 -4996.187} C_VEL
LIN {X 0,Y 516.266,Z 753.461,A -85,B 0,C 180,E1 -4997.745,E2 -4997.745} C_VEL
LIN {X 0,Y 516.327,Z 750.315,A -85,B 0,C 180,E1 -4998.841,E2 -4998.841} C_VEL
LIN {X 0,Y 516.381,Z 746.196,A -85,B 0,C 180,E1 -4999.944,E2 -4999.944} C_VEL
LIN {X 0,Y 516.534,Z 740.954,A -85,B 0,C 180,E1 -5001.057,E2 -5001.057} C_VEL
LIN {X 0,Y 516.641,Z 733.923,A -85,B 0,C 180,E1 -5002.255,E2 -5002.255} C_VEL
LIN {X 0,Y 516.791,Z 728.744,A -85,B 0,C 180,E1 -5003.003,E2 -5003.003} C_VEL
LIN {X 0,Y 517.007,Z 720.586,A -85,B 0,C 180,E1 -5003.99,E2 -5003.99} C_VEL
LIN {X 0,Y 517.284,Z 712.719,A -85,B 0,C 180,E1 -5004.787,E2 -5004.787} C_VEL
LIN {X 0,Y 517.461,Z 704.412,A -85,B 0,C 180,E1 -5005.5,E2 -5005.5} C_VEL
LIN {X 0,Y 517.773,Z 694.74,A -85,B 0,C 180,E1 -5006.185,E2 -5006.185} C_VEL
LIN {X 0,Y 518.003,Z 685.42,A -85,B 0,C 180,E1 -5006.726,E2 -5006.726} C_VEL
LIN {X 0,Y 518.261,Z 676.382,A -85,B 0,C 180,E1 -5007.151,E2 -5007.151} C_VEL
LIN {X 0,Y 518.384,Z 665.666,A -85,B 0,C 180,E1 -5007.54,E2 -5007.54} C_VEL
LIN {X 0,Y 516.483,Z 655.094,A -85,B 0,C 180,E1 -5007.865,E2 -5007.865} C_VEL
LIN {X 0,Y 516.27,Z 653.631,A -85,B 0,C 180,E1 -5007.912,E2 -5007.912} C_VEL
LIN {X 0,Y 516.287,Z 649.028,A -85,B 0,C 180,E1 -5010.656,E2 -5010.656} C_VEL
LIN {X 0,Y 516.37,Z 644.647,A -85,B 0,C 180,E1 -5013.311,E2 -5013.311} C_VEL
LIN {X 0,Y 516.399,Z 638.638,A -85,B 0,C 180,E1 -5016.754,E2 -5016.754} C_VEL
LIN {X 0,Y 516.443,Z 633.14,A -85,B 0,C 180,E1 -5019.88,E2 -5019.88} C_VEL
LIN {X 0,Y 516.498,Z 628.347,A -85,B 0,C 180,E1 -5022.581,E2 -5022.581} C_VEL
LIN {X 0,Y 516.579,Z 623.874,A -85,B 0,C 180,E1 -5025.019,E2 -5025.019} C_VEL
LIN {X 0,Y 516.517,Z 620.15,A -85,B 0,C 180,E1 -5027.026,E2 -5027.026} C_VEL
LIN {X 0,Y 516.857,Z 620.107,A -85,B 0,C 180,E1 -5029.026,E2 -5029.026} C_VEL
LIN {X 0,Y 516.969,Z 620.092,A -85,B 0,C 180,E1 -5031.4,E2 -5031.4} C_VEL
LIN {X 0,Y 517.009,Z 620.087,A -85,B 0,C 180,E1 -5033.757,E2 -5033.757} C_VEL
LIN {X 0,Y 517.082,Z 620.077,A -85,B 0,C 180,E1 -5037.663,E2 -5037.663} C_VEL
LIN {X 0,Y 517.092,Z 620.076,A -85,B 0,C 180,E1 -5040.779,E2 -5040.779} C_VEL
LIN {X 0,Y 517.013,Z 620.086,A -85,B 0,C 180,E1 -5043.117,E2 -5043.117} C_VEL
LIN {X 0,Y 517.007,Z 620.087,A -85,B 0,C 180,E1 -5046.243,E2 -5046.243} C_VEL
LIN {X 0,Y 516.955,Z 620.094,A -85,B 0,C 180,E1 -5049.389,E2 -5049.389} C_VEL
LIN {X 0,Y 516.954,Z 620.093,A -85,B 0,C 180,E1 -5051.81,E2 -5051.81} C_VEL
LIN {X 0,Y 516.94,Z 620.095,A -85,B 0,C 180,E1 -5055.147,E2 -5055.147} C_VEL
LIN {X 0,Y 516.923,Z 620.097,A -85,B 0,C 180,E1 -5058.222,E2 -5058.222} C_VEL
LIN {X 0,Y 516.909,Z 620.099,A -85,B 0,C 180,E1 -5060.702,E2 -5060.702} C_VEL
LIN {X 0,Y 516.908,Z 620.1,A -85,B 0,C 180,E1 -5064.072,E2 -5064.072} C_VEL
LIN {X 0,Y 516.927,Z 620.096,A -85,B 0,C 180,E1 -5066.658,E2 -5066.658} C_VEL
LIN {X 0,Y 516.922,Z 620.097,A -85,B 0,C 180,E1 -5069.527,E2 -5069.527} C_VEL
LIN {X 0,Y 516.898,Z 620.1,A -85,B 0,C 180,E1 -5072.545,E2 -5072.545} C_VEL
LIN {X 0,Y 516.877,Z 620.103,A -85,B 0,C 180,E1 -5075.332,E2 -5075.332} C_VEL
LIN {X 0,Y 516.879,Z 620.101,A -85,B 0,C 180,E1 -5077.944,E2 -5077.944} C_VEL
LIN {X 0,Y 516.883,Z 620.102,A -85,B 0,C 180,E1 -5080.742,E2 -5080.742} C_VEL
LIN {X 0,Y 516.88,Z 620.102,A -85,B 0,C 180,E1 -5082.832,E2 -5082.832} C_VEL
LIN {X 0,Y 516.921,Z 620.097,A -85,B 0,C 180,E1 -5085.011,E2 -5085.011} C_VEL
LIN {X 0,Y 516.914,Z 620.099,A -85,B 0,C 180,E1 -5088.399,E2 -5088.399} C_VEL
LIN {X 0,Y 516.882,Z 620.103,A -85,B 0,C 180,E1 -5091.285,E2 -5091.285} C_VEL
LIN {X 0,Y 516.92,Z 620.281,A -85,B 0,C 180,E1 -5092.28,E2 -5092.28} C_VEL
LIN {X 0,Y 517.606,Z 625.304,A -85,B 0,C 180,E1 -5094.555,E2 -5094.555} C_VEL
LIN {X 0,Y 517.421,Z 631.941,A -85,B 0,C 180,E1 -5097.366,E2 -5097.366} C_VEL
LIN {X 0,Y 517.204,Z 639.413,A -85,B 0,C 180,E1 -5100.42,E2 -5100.42} C_VEL
LIN {X 0,Y 517.042,Z 646.833,A -85,B 0,C 180,E1 -5103.349,E2 -5103.349} C_VEL
LIN {X 0,Y 516.871,Z 654.668,A -85,B 0,C 180,E1 -5106.352,E2 -5106.352} C_VEL
LIN {X 0,Y 516.759,Z 662.526,A -85,B 0,C 180,E1 -5109.293,E2 -5109.293} C_VEL
LIN {X 0,Y 516.607,Z 670.629,A -85,B 0,C 180,E1 -5112.231,E2 -5112.231} C_VEL
LIN {X 0,Y 516.547,Z 678.406,A -85,B 0,C 180,E1 -5115.019,E2 -5115.019} C_VEL
LIN {X 0,Y 516.522,Z 681.443,A -85,B 0,C 180,E1 -5116.1,E2 -5116.1} C_VEL
LIN {X 0,Y 518.461,Z 694.108,A -85,B 0,C 180,E1 -5116.453,E2 -5116.453} C_VEL
LIN {X 0,Y 518.227,Z 707.119,A -85,B 0,C 180,E1 -5116.921,E2 -5116.921} C_VEL
LIN {X 0,Y 517.912,Z 719.422,A -85,B 0,C 180,E1 -5117.531,E2 -5117.531} C_VEL
LIN {X 0,Y 517.659,Z 730.595,A -85,B 0,C 180,E1 -5118.25,E2 -5118.25} C_VEL
LIN {X 0,Y 517.329,Z 741.471,A -85,B 0,C 180,E1 -5119.135,E2 -5119.135} C_VEL
LIN {X 0,Y 517.044,Z 750.336,A -85,B 0,C 180,E1 -5120.02,E2 -5120.02} C_VEL
LIN {X 0,Y 516.813,Z 759.963,A -85,B 0,C 180,E1 -5121.2,E2 -5121.2} C_VEL
LIN {X 0,Y 516.563,Z 767.623,A -85,B 0,C 180,E1 -5122.378,E2 -5122.378} C_VEL
LIN {X 0,Y 516.427,Z 774.681,A -85,B 0,C 180,E1 -5123.75,E2 -5123.75} C_VEL
LIN {X 0,Y 516.313,Z 779.374,A -85,B 0,C 180,E1 -5124.924,E2 -5124.924} C_VEL
LIN {X 0,Y 516.355,Z 782.959,A -85,B 0,C 180,E1 -5126.098,E2 -5126.098} C_VEL
LIN {X 0,Y 516.282,Z 784.807,A -85,B 0,C 180,E1 -5126.879,E2 -5126.879} C_VEL
LIN {X 0,Y 516.261,Z 786.194,A -85,B 0,C 180,E1 -5127.66,E2 -5127.66} C_VEL
LIN {X 0,Y 516.16,Z 787.786,A -85,B 0,C 180,E1 -5129.22,E2 -5129.22} C_VEL
LIN {X 0,Y 516.154,Z 788,A -85,B 0,C 180,E1 -5130,E2 -5130} C_VEL
LIN {X 0,Y 516.192,Z 787.183,A -85,B 0,C 180,E1 -5131.561,E2 -5131.561} C_VEL
LIN {X 0,Y 516.261,Z 786.196,A -85,B 0,C 180,E1 -5132.341,E2 -5132.341} C_VEL
LIN {X 0,Y 516.282,Z 784.809,A -85,B 0,C 180,E1 -5133.122,E2 -5133.122} C_VEL
LIN {X 0,Y 516.344,Z 781.894,A -85,B 0,C 180,E1 -5134.294,E2 -5134.294} C_VEL
LIN {X 0,Y 516.405,Z 777.947,A -85,B 0,C 180,E1 -5135.467,E2 -5135.467} C_VEL
LIN {X 0,Y 516.486,Z 772.032,A -85,B 0,C 180,E1 -5136.808,E2 -5136.808} C_VEL
LIN {X 0,Y 516.641,Z 765.233,A -85,B 0,C 180,E1 -5138.015,E2 -5138.015} C_VEL
LIN {X 0,Y 516.868,Z 756.99,A -85,B 0,C 180,E1 -5139.194,E2 -5139.194} C_VEL
LIN {X 0,Y 517.081,Z 748.537,A -85,B 0,C 180,E1 -5140.177,E2 -5140.177} C_VEL
LIN {X 0,Y 517.441,Z 738.087,A -85,B 0,C 180,E1 -5141.16,E2 -5141.16} C_VEL
LIN {X 0,Y 517.72,Z 726.617,A -85,B 0,C 180,E1 -5142.026,E2 -5142.026} C_VEL
LIN {X 0,Y 517.983,Z 716.399,A -85,B 0,C 180,E1 -5142.638,E2 -5142.638} C_VEL
LIN {X 0,Y 518.273,Z 704.757,A -85,B 0,C 180,E1 -5143.179,E2 -5143.179} C_VEL
LIN {X 0,Y 518.374,Z 692.696,A -85,B 0,C 180,E1 -5143.588,E2 -5143.588} C_VEL
LIN {X 0,Y 516.519,Z 681.428,A -85,B 0,C 180,E1 -5143.901,E2 -5143.901} C_VEL
LIN {X 0,Y 516.571,Z 673.826,A -85,B 0,C 180,E1 -5146.601,E2 -5146.601} C_VEL
LIN {X 0,Y 516.705,Z 665.839,A -85,B 0,C 180,E1 -5149.466,E2 -5149.466} C_VEL
LIN {X 0,Y 516.794,Z 657.816,A -85,B 0,C 180,E1 -5152.382,E2 -5152.382} C_VEL
LIN {X 0,Y 516.943,Z 649.96,A -85,B 0,C 180,E1 -5155.357,E2 -5155.357} C_VEL
LIN {X 0,Y 517.097,Z 643.28,A -85,B 0,C 180,E1 -5157.94,E2 -5157.94} C_VEL
LIN {X 0,Y 517.293,Z 635.432,A -85,B 0,C 180,E1 -5161.083,E2 -5161.083} C_VEL
LIN {X 0,Y 517.482,Z 628.351,A -85,B 0,C 180,E1 -5164.06,E2 -5164.06} C_VEL
LIN {X 0,Y 517.558,Z 624.56,A -85,B 0,C 180,E1 -5165.726,E2 -5165.726} C_VEL
LIN {X 0,Y 516.911,Z 620.095,A -85,B 0,C 180,E1 -5167.878,E2 -5167.878} C_VEL
LIN {X 0,Y 516.887,Z 620.103,A -85,B 0,C 180,E1 -5170.742,E2 -5170.742} C_VEL
LIN {X 0,Y 516.907,Z 620.1,A -85,B 0,C 180,E1 -5172.829,E2 -5172.829} C_VEL
LIN {X 0,Y 516.925,Z 620.097,A -85,B 0,C 180,E1 -5175.01,E2 -5175.01} C_VEL
LIN {X 0,Y 516.917,Z 620.1,A -85,B 0,C 180,E1 -5178.399,E2 -5178.399} C_VEL
LIN {X 0,Y 516.883,Z 620.104,A -85,B 0,C 180,E1 -5181.284,E2 -5181.284} C_VEL
LIN {X 0,Y 516.878,Z 620.104,A -85,B 0,C 180,E1 -5184.22,E2 -5184.22} C_VEL
LIN {X 0,Y 516.898,Z 620.1,A -85,B 0,C 180,E1 -5187.053,E2 -5187.053} C_VEL
LIN {X 0,Y 516.894,Z 620.1,A -85,B 0,C 180,E1 -5189.796,E2 -5189.796} C_VEL
LIN {X 0,Y 516.93,Z 620.098,A -85,B 0,C 180,E1 -5192.467,E2 -5192.467} C_VEL
LIN {X 0,Y 516.913,Z 620.098,A -85,B 0,C 180,E1 -5195.072,E2 -5195.072} C_VEL
LIN {X 0,Y 516.888,Z 620.103,A -85,B 0,C 180,E1 -5198.462,E2 -5198.462} C_VEL
LIN {X 0,Y 516.905,Z 620.099,A -85,B 0,C 180,E1 -5200.955,E2 -5200.955} C_VEL
LIN {X 0,Y 516.916,Z 620.099,A -85,B 0,C 180,E1 -5203.41,E2 -5203.41} C_VEL
LIN {X 0,Y 516.897,Z 620.101,A -85,B 0,C 180,E1 -5205.834,E2 -5205.834} C_VEL
LIN {X 0,Y 516.967,Z 620.091,A -85,B 0,C 180,E1 -5208.234,E2 -5208.234} C_VEL
LIN {X 0,Y 516.972,Z 620.091,A -85,B 0,C 180,E1 -5211.4,E2 -5211.4} C_VEL
LIN {X 0,Y 517.012,Z 620.087,A -85,B 0,C 180,E1 -5213.757,E2 -5213.757} C_VEL
LIN {X 0,Y 517.084,Z 620.078,A -85,B 0,C 180,E1 -5217.663,E2 -5217.663} C_VEL
LIN {X 0,Y 517.097,Z 620.077,A -85,B 0,C 180,E1 -5220.779,E2 -5220.779} C_VEL
LIN {X 0,Y 517.017,Z 620.086,A -85,B 0,C 180,E1 -5223.117,E2 -5223.117} C_VEL
LIN {X 0,Y 517.013,Z 620.086,A -85,B 0,C 180,E1 -5226.243,E2 -5226.243} C_VEL
LIN {X 0,Y 516.957,Z 620.094,A -85,B 0,C 180,E1 -5228.601,E2 -5228.601} C_VEL
LIN {X 0,Y 516.872,Z 620.104,A -85,B 0,C 180,E1 -5229.391,E2 -5229.391} C_VEL
LIN {X 0,Y 516.831,Z 620.697,A -85,B 0,C 180,E1 -5230.182,E2 -5230.182} C_VEL
LIN {X 0,Y 516.781,Z 624.242,A -85,B 0,C 180,E1 -5232.568,E2 -5232.568} C_VEL
LIN {X 0,Y 516.73,Z 628.002,A -85,B 0,C 180,E1 -5235.058,E2 -5235.058} C_VEL
LIN {X 0,Y 516.6,Z 632.894,A -85,B 0,C 180,E1 -5238.234,E2 -5238.234} C_VEL
LIN {X 0,Y 516.522,Z 636.732,A -85,B 0,C 180,E1 -5240.718,E2 -5240.718} C_VEL
LIN {X 0,Y 516.446,Z 640.666,A -85,B 0,C 180,E1 -5243.244,E2 -5243.244} C_VEL
LIN {X 0,Y 516.373,Z 646.195,A -85,B 0,C 180,E1 -5246.689,E2 -5246.689} C_VEL
LIN {X 0,Y 516.276,Z 650.671,A -85,B 0,C 180,E1 -5249.399,E2 -5249.399} C_VEL
LIN {X 0,Y 516.293,Z 653.657,A -85,B 0,C 180,E1 -5251.178,E2 -5251.178} C_VEL
LIN {X 0,Y 518.418,Z 666.646,A -85,B 0,C 180,E1 -5251.576,E2 -5251.576} C_VEL
LIN {X 0,Y 518.159,Z 679.118,A -85,B 0,C 180,E1 -5252.051,E2 -5252.051} C_VEL
LIN {X 0,Y 517.857,Z 690.441,A -85,B 0,C 180,E1 -5252.631,E2 -5252.631} C_VEL
LIN {X 0,Y 517.616,Z 701.473,A -85,B 0,C 180,E1 -5253.36,E2 -5253.36} C_VEL
LIN {X 0,Y 517.26,Z 712.441,A -85,B 0,C 180,E1 -5254.269,E2 -5254.269} C_VEL
LIN {X 0,Y 517.022,Z 721.626,A -85,B 0,C 180,E1 -5255.208,E2 -5255.208} C_VEL
LIN {X 0,Y 516.767,Z 730.152,A -85,B 0,C 180,E1 -5256.271,E2 -5256.271} C_VEL
LIN {X 0,Y 516.541,Z 738.108,A -85,B 0,C 180,E1 -5257.508,E2 -5257.508} C_VEL
LIN {X 0,Y 516.401,Z 744.514,A -85,B 0,C 180,E1 -5258.759,E2 -5258.759} C_VEL
LIN {X 0,Y 516.355,Z 748.647,A -85,B 0,C 180,E1 -5259.77,E2 -5259.77} C_VEL
LIN {X 0,Y 516.289,Z 752.025,A -85,B 0,C 180,E1 -5260.799,E2 -5260.799} C_VEL
LIN {X 0,Y 516.295,Z 754.619,A -85,B 0,C 180,E1 -5261.837,E2 -5261.837} C_VEL
LIN {X 0,Y 516.219,Z 755.872,A -85,B 0,C 180,E1 -5262.521,E2 -5262.521} C_VEL
LIN {X 0,Y 515.529,Z 756.886,A -85,B 0,C 180,E1 -5263.163,E2 -5263.163} C_VEL
LIN {X 0,Y 512.657,Z 757.859,A -85,B 0,C 180,E1 -5264.217,E2 -5264.217} C_VEL
LIN {X 0,Y 510.235,Z 758.035,A -85,B 0,C 180,E1 -5265.07,E2 -5265.07} C_VEL
LIN {X 0,Y 509.187,Z 757.849,A -85,B 0,C 180,E1 -5265.728,E2 -5265.728} C_VEL
LIN {X 0,Y 509.096,Z 757.713,A -85,B 0,C 180,E1 -5265.951,E2 -5265.951} C_VEL
LIN {X 0,Y 509.106,Z 756.169,A -85,B 0,C 180,E1 -5267.435,E2 -5267.435} C_VEL
LIN {X 0,Y 509.171,Z 754.146,A -85,B 0,C 180,E1 -5268.506,E2 -5268.506} C_VEL
LIN {X 0,Y 509.208,Z 751.42,A -85,B 0,C 180,E1 -5269.557,E2 -5269.557} C_VEL
LIN {X 0,Y 509.303,Z 746.878,A -85,B 0,C 180,E1 -5270.859,E2 -5270.859} C_VEL
LIN {X 0,Y 509.452,Z 740.575,A -85,B 0,C 180,E1 -5272.242,E2 -5272.242} C_VEL
LIN {X 0,Y 509.606,Z 734.025,A -85,B 0,C 180,E1 -5273.378,E2 -5273.378} C_VEL
LIN {X 0,Y 509.804,Z 726.642,A -85,B 0,C 180,E1 -5274.425,E2 -5274.425} C_VEL
LIN {X 0,Y 510.14,Z 717.43,A -85,B 0,C 180,E1 -5275.489,E2 -5275.489} C_VEL
LIN {X 0,Y 510.45,Z 707.009,A -85,B 0,C 180,E1 -5276.465,E2 -5276.465} C_VEL
LIN {X 0,Y 510.837,Z 695.92,A -85,B 0,C 180,E1 -5277.295,E2 -5277.295} C_VEL
LIN {X 0,Y 511.133,Z 684.193,A -85,B 0,C 180,E1 -5277.979,E2 -5277.979} C_VEL
LIN {X 0,Y 511.411,Z 671.973,A -85,B 0,C 180,E1 -5278.519,E2 -5278.519} C_VEL
LIN {X 0,Y 511.31,Z 665.536,A -85,B 0,C 180,E1 -5278.747,E2 -5278.747} C_VEL
LIN {X 0,Y 509.21,Z 653.826,A -85,B 0,C 180,E1 -5279.121,E2 -5279.121} C_VEL
LIN {X 0,Y 509.253,Z 649.016,A -85,B 0,C 180,E1 -5282.036,E2 -5282.036} C_VEL
LIN {X 0,Y 509.301,Z 644.76,A -85,B 0,C 180,E1 -5284.673,E2 -5284.673} C_VEL
LIN {X 0,Y 509.379,Z 640.118,A -85,B 0,C 180,E1 -5287.581,E2 -5287.581} C_VEL
LIN {X 0,Y 509.483,Z 635.246,A -85,B 0,C 180,E1 -5290.666,E2 -5290.666} C_VEL
LIN {X 0,Y 509.544,Z 631.339,A -85,B 0,C 180,E1 -5293.163,E2 -5293.163} C_VEL
LIN {X 0,Y 509.648,Z 627.574,A -85,B 0,C 180,E1 -5295.628,E2 -5295.628} C_VEL
LIN {X 0,Y 509.81,Z 622.676,A -85,B 0,C 180,E1 -5298.872,E2 -5298.872} C_VEL
LIN {X 0,Y 509.735,Z 621.504,A -85,B 0,C 180,E1 -5299.674,E2 -5299.674} C_VEL
LIN {X 0,Y 509.792,Z 620.986,A -85,B 0,C 180,E1 -5300.477,E2 -5300.477} C_VEL
LIN {X 0,Y 509.976,Z 620.962,A -85,B 0,C 180,E1 -5302.875,E2 -5302.875} C_VEL
LIN {X 0,Y 509.904,Z 620.971,A -85,B 0,C 180,E1 -5305.256,E2 -5305.256} C_VEL
LIN {X 0,Y 510.06,Z 620.95,A -85,B 0,C 180,E1 -5307.631,E2 -5307.631} C_VEL
LIN {X 0,Y 510.068,Z 620.953,A -85,B 0,C 180,E1 -5310.789,E2 -5310.789} C_VEL
LIN {X 0,Y 509.958,Z 620.965,A -85,B 0,C 180,E1 -5313.16,E2 -5313.16} C_VEL
LIN {X 0,Y 509.959,Z 620.963,A -85,B 0,C 180,E1 -5316.329,E2 -5316.329} C_VEL
LIN {X 0,Y 509.854,Z 620.977,A -85,B 0,C 180,E1 -5318.721,E2 -5318.721} C_VEL
LIN {X 0,Y 509.583,Z 621.055,A -85,B 0,C 180,E1 -5320.73,E2 -5320.73} C_VEL
LIN {X 0,Y 509.48,Z 625.977,A -85,B 0,C 180,E1 -5323.562,E2 -5323.562} C_VEL
LIN {X 0,Y 509.456,Z 630.186,A -85,B 0,C 180,E1 -5326.015,E2 -5326.015} C_VEL
LIN {X 0,Y 509.38,Z 634.448,A -85,B 0,C 180,E1 -5328.501,E2 -5328.501} C_VEL
LIN {X 0,Y 509.314,Z 638.72,A -85,B 0,C 180,E1 -5331.024,E2 -5331.024} C_VEL
LIN {X 0,Y 509.268,Z 643.052,A -85,B 0,C 180,E1 -5333.591,E2 -5333.591} C_VEL
LIN {X 0,Y 509.239,Z 647.494,A -85,B 0,C 180,E1 -5336.225,E2 -5336.225} C_VEL
LIN {X 0,Y 509.177,Z 651.958,A -85,B 0,C 180,E1 -5338.887,E2 -5338.887} C_VEL
LIN {X 0,Y 509.178,Z 653.814,A -85,B 0,C 180,E1 -5339.994,E2 -5339.994} C_VEL
LIN {X 0,Y 511.139,Z 664.667,A -85,B 0,C 180,E1 -5340.322,E2 -5340.322} C_VEL
LIN {X 0,Y 511.503,Z 669.926,A -85,B 0,C 180,E1 -5340.498,E2 -5340.498} C_VEL
LIN {X 0,Y 511.112,Z 682.665,A -85,B 0,C 180,E1 -5341.04,E2 -5341.04} C_VEL
LIN {X 0,Y 510.938,Z 691.335,A -85,B 0,C 180,E1 -5341.512,E2 -5341.512} C_VEL
LIN {X 0,Y 510.574,Z 701.98,A -85,B 0,C 180,E1 -5342.234,E2 -5342.234} C_VEL
LIN {X 0,Y 510.335,Z 710.429,A -85,B 0,C 180,E1 -5342.932,E2 -5342.932} C_VEL
LIN {X 0,Y 510.084,Z 718.104,A -85,B 0,C 180,E1 -5343.68,E2 -5343.68} C_VEL
LIN {X 0,Y 509.868,Z 724.563,A -85,B 0,C 180,E1 -5344.412,E2 -5344.412} C_VEL
LIN {X 0,Y 509.642,Z 731.846,A -85,B 0,C 180,E1 -5345.392,E2 -5345.392} C_VEL
LIN {X 0,Y 509.472,Z 737.988,A -85,B 0,C 180,E1 -5346.382,E2 -5346.382} C_VEL
LIN {X 0,Y 509.364,Z 743.156,A -85,B 0,C 180,E1 -5347.379,E2 -5347.379} C_VEL
LIN {X 0,Y 509.299,Z 747.476,A -85,B 0,C 180,E1 -5348.386,E2 -5348.386} C_VEL
LIN {X 0,Y 509.19,Z 751.061,A -85,B 0,C 180,E1 -5349.412,E2 -5349.412} C_VEL
LIN {X 0,Y 509.111,Z 754.2,A -85,B 0,C 180,E1 -5350.602,E2 -5350.602} C_VEL
LIN {X 0,Y 509.085,Z 756.38,A -85,B 0,C 180,E1 -5351.799,E2 -5351.799} C_VEL
LIN {X 0,Y 509.082,Z 757.619,A -85,B 0,C 180,E1 -5352.972,E2 -5352.972} C_VEL
LIN {X 0,Y 509.093,Z 757.991,A -85,B 0,C 180,E1 -5354.122,E2 -5354.122} C_VEL
LIN {X 0,Y 509.099,Z 757.544,A -85,B 0,C 180,E1 -5355.247,E2 -5355.247} C_VEL
LIN {X 0,Y 509.09,Z 756.311,A -85,B 0,C 180,E1 -5356.35,E2 -5356.35} C_VEL
LIN {X 0,Y 509.128,Z 754.299,A -85,B 0,C 180,E1 -5357.437,E2 -5357.437} C_VEL
LIN {X 0,Y 509.257,Z 750.074,A -85,B 0,C 180,E1 -5358.974,E2 -5358.974} C_VEL
LIN {X 0,Y 509.306,Z 745.936,A -85,B 0,C 180,E1 -5360.084,E2 -5360.084} C_VEL
LIN {X 0,Y 509.463,Z 741.161,A -85,B 0,C 180,E1 -5361.121,E2 -5361.121} C_VEL
LIN {X 0,Y 509.555,Z 734.824,A -85,B 0,C 180,E1 -5362.24,E2 -5362.24} C_VEL
LIN {X 0,Y 509.79,Z 727.979,A -85,B 0,C 180,E1 -5363.237,E2 -5363.237} C_VEL
LIN {X 0,Y 509.966,Z 721.456,A -85,B 0,C 180,E1 -5364.046,E2 -5364.046} C_VEL
LIN {X 0,Y 510.288,Z 713.249,A -85,B 0,C 180,E1 -5364.9,E2 -5364.9} C_VEL
LIN {X 0,Y 510.539,Z 704.223,A -85,B 0,C 180,E1 -5365.684,E2 -5365.684} C_VEL
LIN {X 0,Y 510.848,Z 694.53,A -85,B 0,C 180,E1 -5366.376,E2 -5366.376} C_VEL
LIN {X 0,Y 511.088,Z 685.081,A -85,B 0,C 180,E1 -5366.926,E2 -5366.926} C_VEL
LIN {X 0,Y 511.377,Z 675.307,A -85,B 0,C 180,E1 -5367.38,E2 -5367.38} C_VEL
LIN {X 0,Y 511.456,Z 666.287,A -85,B 0,C 180,E1 -5367.711,E2 -5367.711} C_VEL
LIN {X 0,Y 509.408,Z 655.175,A -85,B 0,C 180,E1 -5368.062,E2 -5368.062} C_VEL
LIN {X 0,Y 509.184,Z 653.776,A -85,B 0,C 180,E1 -5368.104,E2 -5368.104} C_VEL
LIN {X 0,Y 509.213,Z 648.77,A -85,B 0,C 180,E1 -5371.114,E2 -5371.114} C_VEL
LIN {X 0,Y 509.289,Z 644.289,A -85,B 0,C 180,E1 -5373.795,E2 -5373.795} C_VEL
LIN {X 0,Y 509.287,Z 639.726,A -85,B 0,C 180,E1 -5376.41,E2 -5376.41} C_VEL
LIN {X 0,Y 509.368,Z 635.336,A -85,B 0,C 180,E1 -5378.977,E2 -5378.977} C_VEL
LIN {X 0,Y 509.443,Z 629.374,A -85,B 0,C 180,E1 -5382.332,E2 -5382.332} C_VEL
LIN {X 0,Y 509.488,Z 623.402,A -85,B 0,C 180,E1 -5385.623,E2 -5385.623} C_VEL
LIN {X 0,Y 509.469,Z 621.028,A -85,B 0,C 180,E1 -5386.945,E2 -5386.945} C_VEL
LIN {X 0,Y 509.805,Z 620.986,A -85,B 0,C 180,E1 -5388.872,E2 -5388.872} C_VEL
LIN {X 0,Y 509.914,Z 620.971,A -85,B 0,C 180,E1 -5391.28,E2 -5391.28} C_VEL
LIN {X 0,Y 509.976,Z 620.963,A -85,B 0,C 180,E1 -5393.67,E2 -5393.67} C_VEL
LIN {X 0,Y 510.053,Z 620.953,A -85,B 0,C 180,E1 -5397.631,E2 -5397.631} C_VEL
LIN {X 0,Y 510.062,Z 620.951,A -85,B 0,C 180,E1 -5400.789,E2 -5400.789} C_VEL
LIN {X 0,Y 509.956,Z 620.966,A -85,B 0,C 180,E1 -5403.16,E2 -5403.16} C_VEL
LIN {X 0,Y 509.975,Z 620.963,A -85,B 0,C 180,E1 -5406.33,E2 -5406.33} C_VEL
LIN {X 0,Y 509.916,Z 620.97,A -85,B 0,C 180,E1 -5408.72,E2 -5408.72} C_VEL
LIN {X 0,Y 509.901,Z 620.971,A -85,B 0,C 180,E1 -5411.932,E2 -5411.932} C_VEL
LIN {X 0,Y 509.89,Z 620.973,A -85,B 0,C 180,E1 -5415.242,E2 -5415.242} C_VEL
LIN {X 0,Y 509.885,Z 620.974,A -85,B 0,C 180,E1 -5418.001,E2 -5418.001} C_VEL
LIN {X 0,Y 509.847,Z 620.978,A -85,B 0,C 180,E1 -5421.002,E2 -5421.002} C_VEL
LIN {X 0,Y 509.834,Z 620.979,A -85,B 0,C 180,E1 -5423.563,E2 -5423.563} C_VEL
LIN {X 0,Y 509.911,Z 620.97,A -85,B 0,C 180,E1 -5426.38,E2 -5426.38} C_VEL
LIN {X 0,Y 509.883,Z 620.973,A -85,B 0,C 180,E1 -5428.844,E2 -5428.844} C_VEL
LIN {X 0,Y 509.824,Z 620.981,A -85,B 0,C 180,E1 -5431.59,E2 -5431.59} C_VEL
LIN {X 0,Y 509.849,Z 620.979,A -85,B 0,C 180,E1 -5434.414,E2 -5434.414} C_VEL
LIN {X 0,Y 509.816,Z 620.983,A -85,B 0,C 180,E1 -5437.341,E2 -5437.341} C_VEL
LIN {X 0,Y 509.836,Z 620.98,A -85,B 0,C 180,E1 -5440.383,E2 -5440.383} C_VEL
LIN {X 0,Y 509.82,Z 620.982,A -85,B 0,C 180,E1 -5443.063,E2 -5443.063} C_VEL
LIN {X 0,Y 509.829,Z 620.981,A -85,B 0,C 180,E1 -5445.793,E2 -5445.793} C_VEL
LIN {X 0,Y 509.856,Z 620.979,A -85,B 0,C 180,E1 -5448.575,E2 -5448.575} C_VEL
LIN {X 0,Y 509.86,Z 620.978,A -85,B 0,C 180,E1 -5451.786,E2 -5451.786} C_VEL
LIN {X 0,Y 509.915,Z 621.219,A -85,B 0,C 180,E1 -5452.121,E2 -5452.121} C_VEL
LIN {X 0,Y 510.584,Z 625.949,A -85,B 0,C 180,E1 -5454.303,E2 -5454.303} C_VEL
LIN {X 0,Y 510.454,Z 631.216,A -85,B 0,C 180,E1 -5456.584,E2 -5456.584} C_VEL
LIN {X 0,Y 510.233,Z 637.84,A -85,B 0,C 180,E1 -5459.361,E2 -5459.361} C_VEL
LIN {X 0,Y 510.086,Z 644.5,A -85,B 0,C 180,E1 -5462.067,E2 -5462.067} C_VEL
LIN {X 0,Y 509.911,Z 651.212,A -85,B 0,C 180,E1 -5464.706,E2 -5464.706} C_VEL
LIN {X 0,Y 509.776,Z 658.391,A -85,B 0,C 180,E1 -5467.472,E2 -5467.472} C_VEL
LIN {X 0,Y 509.641,Z 665.795,A -85,B 0,C 180,E1 -5470.254,E2 -5470.254} C_VEL
LIN {X 0,Y 509.5,Z 674.871,A -85,B 0,C 180,E1 -5473.575,E2 -5473.575} C_VEL
LIN {X 0,Y 509.468,Z 681.524,A -85,B 0,C 180,E1 -5475.916,E2 -5475.916} C_VEL
LIN {X 0,Y 511.536,Z 694.686,A -85,B 0,C 180,E1 -5476.291,E2 -5476.291} C_VEL
LIN {X 0,Y 511.261,Z 708.026,A -85,B 0,C 180,E1 -5476.79,E2 -5476.79} C_VEL
LIN {X 0,Y 510.926,Z 720.497,A -85,B 0,C 180,E1 -5477.43,E2 -5477.43} C_VEL
LIN {X 0,Y 510.646,Z 731.767,A -85,B 0,C 180,E1 -5478.187,E2 -5478.187} C_VEL
LIN {X 0,Y 510.3,Z 742.444,A -85,B 0,C 180,E1 -5479.084,E2 -5479.084} C_VEL
LIN {X 0,Y 510.01,Z 752.067,A -85,B 0,C 180,E1 -5480.082,E2 -5480.082} C_VEL
LIN {X 0,Y 509.76,Z 759.953,A -85,B 0,C 180,E1 -5481.078,E2 -5481.078} C_VEL
LIN {X 0,Y 509.521,Z 767.623,A -85,B 0,C 180,E1 -5482.272,E2 -5482.272} C_VEL
LIN {X 0,Y 509.336,Z 774.681,A -85,B 0,C 180,E1 -5483.663,E2 -5483.663} C_VEL
LIN {X 0,Y 509.248,Z 779.374,A -85,B 0,C 180,E1 -5484.854,E2 -5484.854} C_VEL
LIN {X 0,Y 509.253,Z 782.959,A -85,B 0,C 180,E1 -5486.044,E2 -5486.044} C_VEL
LIN {X 0,Y 509.2,Z 784.807,A -85,B 0,C 180,E1 -5486.836,E2 -5486.836} C_VEL
LIN {X 0,Y 509.161,Z 786.193,A -85,B 0,C 180,E1 -5487.627,E2 -5487.627} C_VEL
LIN {X 0,Y 509.073,Z 787.785,A -85,B 0,C 180,E1 -5489.209,E2 -5489.209} C_VEL
LIN {X 0,Y 509.065,Z 788,A -85,B 0,C 180,E1 -5490,E2 -5490} C_VEL
LIN {X 0,Y 509.112,Z 787.183,A -85,B 0,C 180,E1 -5491.582,E2 -5491.582} C_VEL
LIN {X 0,Y 509.161,Z 786.195,A -85,B 0,C 180,E1 -5492.374,E2 -5492.374} C_VEL
LIN {X 0,Y 509.201,Z 784.809,A -85,B 0,C 180,E1 -5493.165,E2 -5493.165} C_VEL
LIN {X 0,Y 509.234,Z 781.894,A -85,B 0,C 180,E1 -5494.354,E2 -5494.354} C_VEL
LIN {X 0,Y 509.344,Z 777.947,A -85,B 0,C 180,E1 -5495.543,E2 -5495.543} C_VEL
LIN {X 0,Y 509.41,Z 772.279,A -85,B 0,C 180,E1 -5496.854,E2 -5496.854} C_VEL
LIN {X 0,Y 509.585,Z 765.233,A -85,B 0,C 180,E1 -5498.127,E2 -5498.127} C_VEL
LIN {X 0,Y 509.822,Z 756.962,A -85,B 0,C 180,E1 -5499.322,E2 -5499.322} C_VEL
LIN {X 0,Y 510.065,Z 748.462,A -85,B 0,C 180,E1 -5500.319,E2 -5500.319} C_VEL
LIN {X 0,Y 510.457,Z 737.96,A -85,B 0,C 180,E1 -5501.315,E2 -5501.315} C_VEL
LIN {X 0,Y 510.733,Z 726.433,A -85,B 0,C 180,E1 -5502.194,E2 -5502.194} C_VEL
LIN {X 0,Y 511.024,Z 716.173,A -85,B 0,C 180,E1 -5502.813,E2 -5502.813} C_VEL
LIN {X 0,Y 511.341,Z 704.482,A -85,B 0,C 180,E1 -5503.361,E2 -5503.361} C_VEL
LIN {X 0,Y 511.376,Z 692.842,A -85,B 0,C 180,E1 -5503.765,E2 -5503.765} C_VEL
LIN {X 0,Y 509.433,Z 681.246,A -85,B 0,C 180,E1 -5504.098,E2 -5504.098} C_VEL
LIN {X 0,Y 509.495,Z 673.642,A -85,B 0,C 180,E1 -5506.839,E2 -5506.839} C_VEL
LIN {X 0,Y 509.7,Z 664.509,A -85,B 0,C 180,E1 -5510.164,E2 -5510.164} C_VEL
LIN {X 0,Y 509.746,Z 656.552,A -85,B 0,C 180,E1 -5513.138,E2 -5513.138} C_VEL
LIN {X 0,Y 509.902,Z 649.799,A -85,B 0,C 180,E1 -5515.732,E2 -5515.732} C_VEL
LIN {X 0,Y 510.054,Z 643.723,A -85,B 0,C 180,E1 -5518.133,E2 -5518.133} C_VEL
LIN {X 0,Y 510.201,Z 637.545,A -85,B 0,C 180,E1 -5520.642,E2 -5520.642} C_VEL
LIN {X 0,Y 510.431,Z 630.989,A -85,B 0,C 180,E1 -5523.419,E2 -5523.419} C_VEL
LIN {X 0,Y 510.561,Z 625.852,A -85,B 0,C 180,E1 -5525.693,E2 -5525.693} C_VEL
LIN {X 0,Y 509.851,Z 620.974,A -85,B 0,C 180,E1 -5528.071,E2 -5528.071} C_VEL
LIN {X 0,Y 509.842,Z 620.981,A -85,B 0,C 180,E1 -5530.698,E2 -5530.698} C_VEL
LIN {X 0,Y 509.828,Z 620.982,A -85,B 0,C 180,E1 -5533.571,E2 -5533.571} C_VEL
LIN {X 0,Y 509.821,Z 620.983,A -85,B 0,C 180,E1 -5536.428,E2 -5536.428} C_VEL
LIN {X 0,Y 509.841,Z 620.981,A -85,B 0,C 180,E1 -5539.302,E2 -5539.302} C_VEL
LIN {X 0,Y 509.853,Z 620.978,A -85,B 0,C 180,E1 -5541.786,E2 -5541.786} C_VEL
LIN {X 0,Y 509.838,Z 620.98,A -85,B 0,C 180,E1 -5544.622,E2 -5544.622} C_VEL
LIN {X 0,Y 509.865,Z 620.977,A -85,B 0,C 180,E1 -5547.481,E2 -5547.481} C_VEL
LIN {X 0,Y 509.86,Z 620.977,A -85,B 0,C 180,E1 -5550.274,E2 -5550.274} C_VEL
LIN {X 0,Y 509.887,Z 620.973,A -85,B 0,C 180,E1 -5552.944,E2 -5552.944} C_VEL
LIN {X 0,Y 509.872,Z 620.975,A -85,B 0,C 180,E1 -5555.574,E2 -5555.574} C_VEL
LIN {X 0,Y 509.852,Z 620.977,A -85,B 0,C 180,E1 -5558.998,E2 -5558.998} C_VEL
LIN {X 0,Y 509.89,Z 620.973,A -85,B 0,C 180,E1 -5561.999,E2 -5561.999} C_VEL
LIN {X 0,Y 509.912,Z 620.971,A -85,B 0,C 180,E1 -5564.819,E2 -5564.819} C_VEL
LIN {X 0,Y 509.902,Z 620.971,A -85,B 0,C 180,E1 -5568.124,E2 -5568.124} C_VEL
LIN {X 0,Y 509.918,Z 620.97,A -85,B 0,C 180,E1 -5571.28,E2 -5571.28} C_VEL
LIN {X 0,Y 509.98,Z 620.963,A -85,B 0,C 180,E1 -5573.67,E2 -5573.67} C_VEL
LIN {X 0,Y 510.055,Z 620.953,A -85,B 0,C 180,E1 -5577.631,E2 -5577.631} C_VEL
LIN {X 0,Y 510.067,Z 620.953,A -85,B 0,C 180,E1 -5580.79,E2 -5580.79} C_VEL
LIN {X 0,Y 509.959,Z 620.965,A -85,B 0,C 180,E1 -5583.16,E2 -5583.16} C_VEL
LIN {X 0,Y 509.981,Z 620.962,A -85,B 0,C 180,E1 -5586.33,E2 -5586.33} C_VEL
LIN {X 0,Y 509.895,Z 620.974,A -85,B 0,C 180,E1 -5588.721,E2 -5588.721} C_VEL
LIN {X 0,Y 509.813,Z 620.984,A -85,B 0,C 180,E1 -5589.522,E2 -5589.522} C_VEL
LIN {X 0,Y 509.831,Z 622.991,A -85,B 0,C 180,E1 -5591.127,E2 -5591.127} C_VEL
LIN {X 0,Y 509.666,Z 627.792,A -85,B 0,C 180,E1 -5594.372,E2 -5594.372} C_VEL
LIN {X 0,Y 509.574,Z 632.772,A -85,B 0,C 180,E1 -5597.663,E2 -5597.663} C_VEL
LIN {X 0,Y 509.499,Z 636.825,A -85,B 0,C 180,E1 -5600.284,E2 -5600.284} C_VEL
LIN {X 0,Y 509.394,Z 640.602,A -85,B 0,C 180,E1 -5602.725,E2 -5602.725} C_VEL
LIN {X 0,Y 509.318,Z 644.683,A -85,B 0,C 180,E1 -5605.326,E2 -5605.326} C_VEL
LIN {X 0,Y 509.28,Z 648.953,A -85,B 0,C 180,E1 -5607.982,E2 -5607.982} C_VEL
LIN {X 0,Y 509.226,Z 653.886,A -85,B 0,C 180,E1 -5610.977,E2 -5610.977} C_VEL
LIN {X 0,Y 511.513,Z 667.318,A -85,B 0,C 180,E1 -5611.408,E2 -5611.408} C_VEL
LIN {X 0,Y 511.244,Z 680.104,A -85,B 0,C 180,E1 -5611.909,E2 -5611.909} C_VEL
LIN {X 0,Y 510.904,Z 691.782,A -85,B 0,C 180,E1 -5612.53,E2 -5612.53} C_VEL
LIN {X 0,Y 510.621,Z 702.554,A -85,B 0,C 180,E1 -5613.269,E2 -5613.269} C_VEL
LIN {X 0,Y 510.307,Z 712.155,A -85,B 0,C 180,E1 -5614.08,E2 -5614.08} C_VEL
LIN {X 0,Y 510.013,Z 722.189,A -85,B 0,C 180,E1 -5615.122,E2 -5615.122} C_VEL
LIN {X 0,Y 509.719,Z 730.278,A -85,B 0,C 180,E1 -5616.154,E2 -5616.154} C_VEL
LIN {X 0,Y 509.495,Z 737.968,A -85,B 0,C 180,E1 -5617.369,E2 -5617.369} C_VEL
LIN {X 0,Y 509.36,Z 744.351,A -85,B 0,C 180,E1 -5618.632,E2 -5618.632} C_VEL
LIN {X 0,Y 509.238,Z 749.458,A -85,B 0,C 180,E1 -5619.922,E2 -5619.922} C_VEL
LIN {X 0,Y 509.213,Z 752.783,A -85,B 0,C 180,E1 -5621.022,E2 -5621.022} C_VEL
LIN {X 0,Y 509.196,Z 754.668,A -85,B 0,C 180,E1 -5621.814,E2 -5621.814} C_VEL
LIN {X 0,Y 509.106,Z 756.627,A -85,B 0,C 180,E1 -5622.976,E2 -5622.976} C_VEL
LIN {X 0,Y 509.1,Z 757.706,A -85,B 0,C 180,E1 -5624.123,E2 -5624.123} C_VEL
LIN {X 0,Y 509.103,Z 757.965,A -85,B 0,C 180,E1 -5625.248,E2 -5625.248} C_VEL
LIN {X 0,Y 509.096,Z 757.713,A -85,B 0,C 180,E1 -5625.951,E2 -5625.951} C_VEL
LIN {X 0,Y 508.42,Z 757.215,A -85,B 0,C 180,E1 -5626.609,E2 -5626.609} C_VEL
LIN {X 0,Y 505.586,Z 755.883,A -85,B 0,C 180,E1 -5627.671,E2 -5627.671} C_VEL
LIN {X 0,Y 503.205,Z 754.343,A -85,B 0,C 180,E1 -5628.517,E2 -5628.517} C_VEL
LIN {X 0,Y 502.19,Z 752.854,A -85,B 0,C 180,E1 -5629.162,E2 -5629.162} C_VEL
LIN {X 0,Y 502.111,Z 752.277,A -85,B 0,C 180,E1 -5629.379,E2 -5629.379} C_VEL
LIN {X 0,Y 502.228,Z 748.183,A -85,B 0,C 180,E1 -5630.655,E2 -5630.655} C_VEL
LIN {X 0,Y 502.347,Z 742.442,A -85,B 0,C 180,E1 -5632.006,E2 -5632.006} C_VEL
LIN {X 0,Y 502.547,Z 735.491,A -85,B 0,C 180,E1 -5633.284,E2 -5633.284} C_VEL
LIN {X 0,Y 502.79,Z 726.927,A -85,B 0,C 180,E1 -5634.543,E2 -5634.543} C_VEL
LIN {X 0,Y 503.129,Z 717.522,A -85,B 0,C 180,E1 -5635.644,E2 -5635.644} C_VEL
LIN {X 0,Y 503.48,Z 707.452,A -85,B 0,C 180,E1 -5636.6,E2 -5636.6} C_VEL
LIN {X 0,Y 503.87,Z 697.002,A -85,B 0,C 180,E1 -5637.402,E2 -5637.402} C_VEL
LIN {X 0,Y 504.199,Z 685.73,A -85,B 0,C 180,E1 -5638.088,E2 -5638.088} C_VEL
LIN {X 0,Y 504.505,Z 672.866,A -85,B 0,C 180,E1 -5638.677,E2 -5638.677} C_VEL
LIN {X 0,Y 504.478,Z 666.783,A -85,B 0,C 180,E1 -5638.898,E2 -5638.898} C_VEL
LIN {X 0,Y 502.124,Z 654.03,A -85,B 0,C 180,E1 -5639.322,E2 -5639.322} C_VEL
LIN {X 0,Y 502.179,Z 648.88,A -85,B 0,C 180,E1 -5642.494,E2 -5642.494} C_VEL
LIN {X 0,Y 502.237,Z 644.143,A -85,B 0,C 180,E1 -5645.447,E2 -5645.447} C_VEL
LIN {X 0,Y 502.325,Z 640.423,A -85,B 0,C 180,E1 -5647.805,E2 -5647.805} C_VEL
LIN {X 0,Y 502.406,Z 636.386,A -85,B 0,C 180,E1 -5650.383,E2 -5650.383} C_VEL
LIN {X 0,Y 502.476,Z 632.469,A -85,B 0,C 180,E1 -5652.919,E2 -5652.919} C_VEL
LIN {X 0,Y 502.593,Z 628.666,A -85,B 0,C 180,E1 -5655.421,E2 -5655.421} C_VEL
LIN {X 0,Y 502.756,Z 623.758,A -85,B 0,C 180,E1 -5658.714,E2 -5658.714} C_VEL
LIN {X 0,Y 502.693,Z 622.572,A -85,B 0,C 180,E1 -5659.528,E2 -5659.528} C_VEL
LIN {X 0,Y 502.742,Z 621.864,A -85,B 0,C 180,E1 -5660.343,E2 -5660.343} C_VEL
LIN {X 0,Y 502.941,Z 621.839,A -85,B 0,C 180,E1 -5662.814,E2 -5662.814} C_VEL
LIN {X 0,Y 502.873,Z 621.847,A -85,B 0,C 180,E1 -5665.19,E2 -5665.19} C_VEL
LIN {X 0,Y 503.029,Z 621.825,A -85,B 0,C 180,E1 -5667.597,E2 -5667.597} C_VEL
LIN {X 0,Y 503.032,Z 621.826,A -85,B 0,C 180,E1 -5670,E2 -5670} C_VEL
LIN {X 0,Y 503.029,Z 621.827,A -85,B 0,C 180,E1 -5672.402,E2 -5672.402} C_VEL
LIN {X 0,Y 502.937,Z 621.838,A -85,B 0,C 180,E1 -5675.613,E2 -5675.613} C_VEL
LIN {X 0,Y 502.87,Z 621.847,A -85,B 0,C 180,E1 -5678.033,E2 -5678.033} C_VEL
LIN {X 0,Y 502.515,Z 622.008,A -85,B 0,C 180,E1 -5680.883,E2 -5680.883} C_VEL
LIN {X 0,Y 502.441,Z 628.37,A -85,B 0,C 180,E1 -5684.582,E2 -5684.582} C_VEL
LIN {X 0,Y 502.34,Z 634.058,A -85,B 0,C 180,E1 -5687.926,E2 -5687.926} C_VEL
LIN {X 0,Y 502.265,Z 638.386,A -85,B 0,C 180,E1 -5690.476,E2 -5690.476} C_VEL
LIN {X 0,Y 502.202,Z 642.728,A -85,B 0,C 180,E1 -5693.069,E2 -5693.069} C_VEL
LIN {X 0,Y 502.149,Z 647.161,A -85,B 0,C 180,E1 -5695.713,E2 -5695.713} C_VEL
LIN {X 0,Y 502.094,Z 651.683,A -85,B 0,C 180,E1 -5698.418,E2 -5698.418} C_VEL
LIN {X 0,Y 502.109,Z 653.992,A -85,B 0,C 180,E1 -5699.794,E2 -5699.794} C_VEL
LIN {X 0,Y 504.218,Z 665.152,A -85,B 0,C 180,E1 -5700.142,E2 -5700.142} C_VEL
LIN {X 0,Y 504.603,Z 670.576,A -85,B 0,C 180,E1 -5700.33,E2 -5700.33} C_VEL
LIN {X 0,Y 504.216,Z 682.695,A -85,B 0,C 180,E1 -5700.853,E2 -5700.853} C_VEL
LIN {X 0,Y 503.981,Z 692.001,A -85,B 0,C 180,E1 -5701.371,E2 -5701.371} C_VEL
LIN {X 0,Y 503.652,Z 701.53,A -85,B 0,C 180,E1 -5702.022,E2 -5702.022} C_VEL
LIN {X 0,Y 503.366,Z 710.346,A -85,B 0,C 180,E1 -5702.753,E2 -5702.753} C_VEL
LIN {X 0,Y 503.054,Z 718.996,A -85,B 0,C 180,E1 -5703.615,E2 -5703.615} C_VEL
LIN {X 0,Y 502.81,Z 726.023,A -85,B 0,C 180,E1 -5704.445,E2 -5704.445} C_VEL
LIN {X 0,Y 502.577,Z 732.746,A -85,B 0,C 180,E1 -5705.383,E2 -5705.383} C_VEL
LIN {X 0,Y 502.405,Z 739.262,A -85,B 0,C 180,E1 -5706.478,E2 -5706.478} C_VEL
LIN {X 0,Y 502.275,Z 744.39,A -85,B 0,C 180,E1 -5707.524,E2 -5707.524} C_VEL
LIN {X 0,Y 502.193,Z 749,A -85,B 0,C 180,E1 -5708.689,E2 -5708.689} C_VEL
LIN {X 0,Y 502.044,Z 753.208,A -85,B 0,C 180,E1 -5710.086,E2 -5710.086} C_VEL
LIN {X 0,Y 501.984,Z 755.476,A -85,B 0,C 180,E1 -5711.148,E2 -5711.148} C_VEL
LIN {X 0,Y 501.985,Z 757.035,A -85,B 0,C 180,E1 -5712.222,E2 -5712.222} C_VEL
LIN {X 0,Y 501.989,Z 757.892,A -85,B 0,C 180,E1 -5713.315,E2 -5713.315} C_VEL
LIN {X 0,Y 502.008,Z 758.017,A -85,B 0,C 180,E1 -5714.439,E2 -5714.439} C_VEL
LIN {X 0,Y 502.009,Z 757.364,A -85,B 0,C 180,E1 -5715.574,E2 -5715.574} C_VEL
LIN {X 0,Y 501.997,Z 755.898,A -85,B 0,C 180,E1 -5716.718,E2 -5716.718} C_VEL
LIN {X 0,Y 502.092,Z 753.516,A -85,B 0,C 180,E1 -5717.89,E2 -5717.89} C_VEL
LIN {X 0,Y 502.19,Z 750.107,A -85,B 0,C 180,E1 -5719.087,E2 -5719.087} C_VEL
LIN {X 0,Y 502.262,Z 745.492,A -85,B 0,C 180,E1 -5720.317,E2 -5720.317} C_VEL
LIN {X 0,Y 502.396,Z 740.899,A -85,B 0,C 180,E1 -5721.308,E2 -5721.308} C_VEL
LIN {X 0,Y 502.553,Z 734.344,A -85,B 0,C 180,E1 -5722.461,E2 -5722.461} C_VEL
LIN {X 0,Y 502.769,Z 728.654,A -85,B 0,C 180,E1 -5723.303,E2 -5723.303} C_VEL
LIN {X 0,Y 502.945,Z 722.048,A -85,B 0,C 180,E1 -5724.141,E2 -5724.141} C_VEL
LIN {X 0,Y 503.273,Z 713.228,A -85,B 0,C 180,E1 -5725.072,E2 -5725.072} C_VEL
LIN {X 0,Y 503.602,Z 704.285,A -85,B 0,C 180,E1 -5725.855,E2 -5725.855} C_VEL
LIN {X 0,Y 503.938,Z 694.232,A -85,B 0,C 180,E1 -5726.578,E2 -5726.578} C_VEL
LIN {X 0,Y 504.232,Z 683.604,A -85,B 0,C 180,E1 -5727.191,E2 -5727.191} C_VEL
LIN {X 0,Y 504.534,Z 672.49,A -85,B 0,C 180,E1 -5727.686,E2 -5727.686} C_VEL
LIN {X 0,Y 504.469,Z 666.931,A -85,B 0,C 180,E1 -5727.888,E2 -5727.888} C_VEL
LIN {X 0,Y 502.293,Z 655.085,A -85,B 0,C 180,E1 -5728.268,E2 -5728.268} C_VEL
LIN {X 0,Y 502.132,Z 653.944,A -85,B 0,C 180,E1 -5728.334,E2 -5728.334} C_VEL
LIN {X 0,Y 502.182,Z 648.096,A -85,B 0,C 180,E1 -5731.844,E2 -5731.844} C_VEL
LIN {X 0,Y 502.189,Z 643.971,A -85,B 0,C 180,E1 -5734.289,E2 -5734.289} C_VEL
LIN {X 0,Y 502.266,Z 638.567,A -85,B 0,C 180,E1 -5737.443,E2 -5737.443} C_VEL
LIN {X 0,Y 502.293,Z 633.431,A -85,B 0,C 180,E1 -5740.378,E2 -5740.378} C_VEL
LIN {X 0,Y 502.347,Z 628.982,A -85,B 0,C 180,E1 -5742.914,E2 -5742.914} C_VEL
LIN {X 0,Y 502.426,Z 624.434,A -85,B 0,C 180,E1 -5745.417,E2 -5745.417} C_VEL
LIN {X 0,Y 502.398,Z 621.909,A -85,B 0,C 180,E1 -5746.861,E2 -5746.861} C_VEL
LIN {X 0,Y 502.758,Z 621.864,A -85,B 0,C 180,E1 -5748.714,E2 -5748.714} C_VEL
LIN {X 0,Y 502.899,Z 621.846,A -85,B 0,C 180,E1 -5751.967,E2 -5751.967} C_VEL
LIN {X 0,Y 502.937,Z 621.84,A -85,B 0,C 180,E1 -5754.386,E2 -5754.386} C_VEL
LIN {X 0,Y 503.022,Z 621.828,A -85,B 0,C 180,E1 -5757.598,E2 -5757.598} C_VEL
LIN {X 0,Y 503.023,Z 621.829,A -85,B 0,C 180,E1 -5760,E2 -5760} C_VEL
LIN {X 0,Y 503.021,Z 621.83,A -85,B 0,C 180,E1 -5762.402,E2 -5762.402} C_VEL
LIN {X 0,Y 502.936,Z 621.84,A -85,B 0,C 180,E1 -5765.614,E2 -5765.614} C_VEL
LIN {X 0,Y 502.899,Z 621.843,A -85,B 0,C 180,E1 -5768.033,E2 -5768.033} C_VEL
LIN {X 0,Y 502.878,Z 621.846,A -85,B 0,C 180,E1 -5771.283,E2 -5771.283} C_VEL
LIN {X 0,Y 502.842,Z 621.851,A -85,B 0,C 180,E1 -5774.571,E2 -5774.571} C_VEL
LIN {X 0,Y 502.859,Z 621.85,A -85,B 0,C 180,E1 -5777.907,E2 -5777.907} C_VEL
LIN {X 0,Y 502.825,Z 621.853,A -85,B 0,C 180,E1 -5780.536,E2 -5780.536} C_VEL
LIN {X 0,Y 502.794,Z 621.858,A -85,B 0,C 180,E1 -5783.041,E2 -5783.041} C_VEL
LIN {X 0,Y 502.839,Z 621.851,A -85,B 0,C 180,E1 -5785.676,E2 -5785.676} C_VEL
LIN {X 0,Y 502.84,Z 621.85,A -85,B 0,C 180,E1 -5788.373,E2 -5788.373} C_VEL
LIN {X 0,Y 502.795,Z 621.857,A -85,B 0,C 180,E1 -5791.5,E2 -5791.5} C_VEL
LIN {X 0,Y 502.802,Z 621.857,A -85,B 0,C 180,E1 -5794.445,E2 -5794.445} C_VEL
LIN {X 0,Y 502.778,Z 621.86,A -85,B 0,C 180,E1 -5797.179,E2 -5797.179} C_VEL
LIN {X 0,Y 502.786,Z 621.857,A -85,B 0,C 180,E1 -5800.016,E2 -5800.016} C_VEL
LIN {X 0,Y 502.8,Z 621.855,A -85,B 0,C 180,E1 -5802.2,E2 -5802.2} C_VEL
LIN {X 0,Y 502.799,Z 621.858,A -85,B 0,C 180,E1 -5805.469,E2 -5805.469} C_VEL
LIN {X 0,Y 502.819,Z 621.855,A -85,B 0,C 180,E1 -5808.935,E2 -5808.935} C_VEL
LIN {X 0,Y 502.833,Z 621.925,A -85,B 0,C 180,E1 -5811.851,E2 -5811.851} C_VEL
LIN {X 0,Y 503.553,Z 626.747,A -85,B 0,C 180,E1 -5814.114,E2 -5814.114} C_VEL
LIN {X 0,Y 503.509,Z 631.144,A -85,B 0,C 180,E1 -5816.061,E2 -5816.061} C_VEL
LIN {X 0,Y 503.25,Z 637.768,A -85,B 0,C 180,E1 -5818.889,E2 -5818.889} C_VEL
LIN {X 0,Y 503.088,Z 644.432,A -85,B 0,C 180,E1 -5821.654,E2 -5821.654} C_VEL
LIN {X 0,Y 502.862,Z 652.208,A -85,B 0,C 180,E1 -5824.77,E2 -5824.77} C_VEL
LIN {X 0,Y 502.68,Z 660.05,A -85,B 0,C 180,E1 -5827.822,E2 -5827.822} C_VEL
LIN {X 0,Y 502.556,Z 666.769,A -85,B 0,C 180,E1 -5830.39,E2 -5830.39} C_VEL
LIN {X 0,Y 502.437,Z 675.801,A -85,B 0,C 180,E1 -5833.755,E2 -5833.755} C_VEL
LIN {X 0,Y 502.378,Z 681.254,A -85,B 0,C 180,E1 -5835.713,E2 -5835.713} C_VEL
LIN {X 0,Y 504.567,Z 694.428,A -85,B 0,C 180,E1 -5836.098,E2 -5836.098} C_VEL
LIN {X 0,Y 504.342,Z 707.776,A -85,B 0,C 180,E1 -5836.605,E2 -5836.605} C_VEL
LIN {X 0,Y 503.961,Z 720.527,A -85,B 0,C 180,E1 -5837.27,E2 -5837.27} C_VEL
LIN {X 0,Y 503.665,Z 731.528,A -85,B 0,C 180,E1 -5838.021,E2 -5838.021} C_VEL
LIN {X 0,Y 503.305,Z 742.21,A -85,B 0,C 180,E1 -5838.931,E2 -5838.931} C_VEL
LIN {X 0,Y 502.969,Z 751.836,A -85,B 0,C 180,E1 -5839.941,E2 -5839.941} C_VEL
LIN {X 0,Y 502.697,Z 759.727,A -85,B 0,C 180,E1 -5840.951,E2 -5840.951} C_VEL
LIN {X 0,Y 502.449,Z 767.434,A -85,B 0,C 180,E1 -5842.162,E2 -5842.162} C_VEL
LIN {X 0,Y 502.255,Z 774.536,A -85,B 0,C 180,E1 -5843.573,E2 -5843.573} C_VEL
LIN {X 0,Y 502.185,Z 779.261,A -85,B 0,C 180,E1 -5844.781,E2 -5844.781} C_VEL
LIN {X 0,Y 502.15,Z 782.871,A -85,B 0,C 180,E1 -5845.988,E2 -5845.988} C_VEL
LIN {X 0,Y 502.121,Z 784.732,A -85,B 0,C 180,E1 -5846.791,E2 -5846.791} C_VEL
LIN {X 0,Y 502.035,Z 787.122,A -85,B 0,C 180,E1 -5848.396,E2 -5848.396} C_VEL
LIN {X 0,Y 501.98,Z 787.945,A -85,B 0,C 180,E1 -5850,E2 -5850} C_VEL
LIN {X 0,Y 502.035,Z 787.122,A -85,B 0,C 180,E1 -5851.605,E2 -5851.605} C_VEL
LIN {X 0,Y 502.066,Z 786.128,A -85,B 0,C 180,E1 -5852.407,E2 -5852.407} C_VEL
LIN {X 0,Y 502.121,Z 784.732,A -85,B 0,C 180,E1 -5853.21,E2 -5853.21} C_VEL
LIN {X 0,Y 502.126,Z 781.794,A -85,B 0,C 180,E1 -5854.415,E2 -5854.415} C_VEL
LIN {X 0,Y 502.259,Z 777.819,A -85,B 0,C 180,E1 -5855.621,E2 -5855.621} C_VEL
LIN {X 0,Y 502.336,Z 771.801,A -85,B 0,C 180,E1 -5857.012,E2 -5857.012} C_VEL
LIN {X 0,Y 502.516,Z 765.013,A -85,B 0,C 180,E1 -5858.242,E2 -5858.242} C_VEL
LIN {X 0,Y 502.782,Z 756.714,A -85,B 0,C 180,E1 -5859.454,E2 -5859.454} C_VEL
LIN {X 0,Y 503.059,Z 748.205,A -85,B 0,C 180,E1 -5860.464,E2 -5860.464} C_VEL
LIN {X 0,Y 503.49,Z 737.694,A -85,B 0,C 180,E1 -5861.473,E2 -5861.473} C_VEL
LIN {X 0,Y 503.768,Z 726.159,A -85,B 0,C 180,E1 -5862.365,E2 -5862.365} C_VEL
LIN {X 0,Y 504.075,Z 715.89,A -85,B 0,C 180,E1 -5862.993,E2 -5862.993} C_VEL
LIN {X 0,Y 504.412,Z 704.184,A -85,B 0,C 180,E1 -5863.548,E2 -5863.548} C_VEL
LIN {X 0,Y 504.423,Z 693.422,A -85,B 0,C 180,E1 -5863.933,E2 -5863.933} C_VEL
LIN {X 0,Y 502.341,Z 681.011,A -85,B 0,C 180,E1 -5864.301,E2 -5864.301} C_VEL
LIN {X 0,Y 502.445,Z 673.459,A -85,B 0,C 180,E1 -5867.082,E2 -5867.082} C_VEL
LIN {X 0,Y 502.618,Z 664.295,A -85,B 0,C 180,E1 -5870.471,E2 -5870.471} C_VEL
LIN {X 0,Y 502.697,Z 656.409,A -85,B 0,C 180,E1 -5873.481,E2 -5873.481} C_VEL
LIN {X 0,Y 502.883,Z 649.649,A -85,B 0,C 180,E1 -5876.118,E2 -5876.118} C_VEL
LIN {X 0,Y 503.058,Z 642.983,A -85,B 0,C 180,E1 -5878.815,E2 -5878.815} C_VEL
LIN {X 0,Y 503.322,Z 635.277,A -85,B 0,C 180,E1 -5882.046,E2 -5882.046} C_VEL
LIN {X 0,Y 503.568,Z 628.791,A -85,B 0,C 180,E1 -5884.905,E2 -5884.905} C_VEL
LIN {X 0,Y 503.277,Z 624.544,A -85,B 0,C 180,E1 -5886.904,E2 -5886.904} C_VEL
LIN {X 0,Y 502.843,Z 621.847,A -85,B 0,C 180,E1 -5888.289,E2 -5888.289} C_VEL
LIN {X 0,Y 502.823,Z 621.856,A -85,B 0,C 180,E1 -5891.066,E2 -5891.066} C_VEL
LIN {X 0,Y 502.784,Z 621.86,A -85,B 0,C 180,E1 -5893.376,E2 -5893.376} C_VEL
LIN {X 0,Y 502.792,Z 621.857,A -85,B 0,C 180,E1 -5895.661,E2 -5895.661} C_VEL
LIN {X 0,Y 502.821,Z 621.855,A -85,B 0,C 180,E1 -5899.005,E2 -5899.005} C_VEL
LIN {X 0,Y 502.795,Z 621.857,A -85,B 0,C 180,E1 -5902.046,E2 -5902.046} C_VEL
LIN {X 0,Y 502.806,Z 621.855,A -85,B 0,C 180,E1 -5905.035,E2 -5905.035} C_VEL
LIN {X 0,Y 502.787,Z 621.857,A -85,B 0,C 180,E1 -5907.916,E2 -5907.916} C_VEL
LIN {X 0,Y 502.826,Z 621.853,A -85,B 0,C 180,E1 -5910.712,E2 -5910.712} C_VEL
LIN {X 0,Y 502.864,Z 621.849,A -85,B 0,C 180,E1 -5913.439,E2 -5913.439} C_VEL
LIN {X 0,Y 502.793,Z 621.855,A -85,B 0,C 180,E1 -5916.086,E2 -5916.086} C_VEL
LIN {X 0,Y 502.785,Z 621.859,A -85,B 0,C 180,E1 -5918.689,E2 -5918.689} C_VEL
LIN {X 0,Y 502.832,Z 621.852,A -85,B 0,C 180,E1 -5921.248,E2 -5921.248} C_VEL
LIN {X 0,Y 502.824,Z 621.854,A -85,B 0,C 180,E1 -5923.767,E2 -5923.767} C_VEL
LIN {X 0,Y 502.833,Z 621.852,A -85,B 0,C 180,E1 -5926.255,E2 -5926.255} C_VEL
LIN {X 0,Y 502.879,Z 621.848,A -85,B 0,C 180,E1 -5928.717,E2 -5928.717} C_VEL
LIN {X 0,Y 502.904,Z 621.842,A -85,B 0,C 180,E1 -5931.967,E2 -5931.967} C_VEL
LIN {X 0,Y 502.94,Z 621.838,A -85,B 0,C 180,E1 -5934.387,E2 -5934.387} C_VEL
LIN {X 0,Y 503.025,Z 621.829,A -85,B 0,C 180,E1 -5937.598,E2 -5937.598} C_VEL
LIN {X 0,Y 503.028,Z 621.828,A -85,B 0,C 180,E1 -5940,E2 -5940} C_VEL
LIN {X 0,Y 503.027,Z 621.829,A -85,B 0,C 180,E1 -5942.402,E2 -5942.402} C_VEL
LIN {X 0,Y 502.942,Z 621.84,A -85,B 0,C 180,E1 -5945.614,E2 -5945.614} C_VEL
LIN {X 0,Y 502.899,Z 621.846,A -85,B 0,C 180,E1 -5948.033,E2 -5948.033} C_VEL
LIN {X 0,Y 502.768,Z 621.862,A -85,B 0,C 180,E1 -5949.657,E2 -5949.657} C_VEL
LIN {X 0,Y 502.731,Z 625.32,A -85,B 0,C 180,E1 -5952.105,E2 -5952.105} C_VEL
LIN {X 0,Y 502.601,Z 630.187,A -85,B 0,C 180,E1 -5955.408,E2 -5955.408} C_VEL
LIN {X 0,Y 502.485,Z 635.227,A -85,B 0,C 180,E1 -5958.765,E2 -5958.765} C_VEL
LIN {X 0,Y 502.366,Z 639.163,A -85,B 0,C 180,E1 -5961.33,E2 -5961.33} C_VEL
LIN {X 0,Y 502.267,Z 643.224,A -85,B 0,C 180,E1 -5963.94,E2 -5963.94} C_VEL
LIN {X 0,Y 502.245,Z 647.387,A -85,B 0,C 180,E1 -5966.602,E2 -5966.602} C_VEL
LIN {X 0,Y 502.127,Z 651.773,A -85,B 0,C 180,E1 -5969.333,E2 -5969.333} C_VEL
LIN {X 0,Y 502.123,Z 654.133,A -85,B 0,C 180,E1 -5970.781,E2 -5970.781} C_VEL
LIN {X 0,Y 504.511,Z 667.043,A -85,B 0,C 180,E1 -5971.2,E2 -5971.2} C_VEL
LIN {X 0,Y 504.341,Z 679.701,A -85,B 0,C 180,E1 -5971.7,E2 -5971.7} C_VEL
LIN {X 0,Y 503.983,Z 691.919,A -85,B 0,C 180,E1 -5972.353,E2 -5972.353} C_VEL
LIN {X 0,Y 503.662,Z 703.333,A -85,B 0,C 180,E1 -5973.151,E2 -5973.151} C_VEL
LIN {X 0,Y 503.296,Z 713.678,A -85,B 0,C 180,E1 -5974.053,E2 -5974.053} C_VEL
LIN {X 0,Y 502.994,Z 723.152,A -85,B 0,C 180,E1 -5975.073,E2 -5975.073} C_VEL
LIN {X 0,Y 502.671,Z 731.674,A -85,B 0,C 180,E1 -5976.208,E2 -5976.208} C_VEL
LIN {X 0,Y 502.412,Z 739.652,A -85,B 0,C 180,E1 -5977.53,E2 -5977.53} C_VEL
LIN {X 0,Y 502.288,Z 745.222,A -85,B 0,C 180,E1 -5978.691,E2 -5978.691} C_VEL
LIN {X 0,Y 502.148,Z 750.401,A -85,B 0,C 180,E1 -5980.077,E2 -5980.077} C_VEL
LIN {X 0,Y 502.127,Z 754.494,A -85,B 0,C 180,E1 -5981.616,E2 -5981.616} C_VEL
LIN {X 0,Y 502.055,Z 755.662,A -85,B 0,C 180,E1 -5982.216,E2 -5982.216} C_VEL
LIN {X 0,Y 501.999,Z 757.207,A -85,B 0,C 180,E1 -5983.315,E2 -5983.315} C_VEL
LIN {X 0,Y 502.012,Z 758.028,A -85,B 0,C 180,E1 -5984.44,E2 -5984.44} C_VEL
LIN {X 0,Y 502.014,Z 758.042,A -85,B 0,C 180,E1 -5985.574,E2 -5985.574} C_VEL
LIN {X 0,Y 501.999,Z 757.258,A -85,B 0,C 180,E1 -5986.719,E2 -5986.719} C_VEL
LIN {X 0,Y 502.048,Z 755.614,A -85,B 0,C 180,E1 -5987.896,E2 -5987.896} C_VEL
LIN {X 0,Y 502.111,Z 752.277,A -85,B 0,C 180,E1 -5989.379,E2 -5989.379} C_VEL
LIN {X 0,Y 501.461,Z 750.485,A -85,B 0,C 180,E1 -5990.018,E2 -5990.018} C_VEL
LIN {X 0,Y 498.668,Z 747.12,A -85,B 0,C 180,E1 -5991.041,E2 -5991.041} C_VEL
LIN {X 0,Y 495.925,Z 743.01,A -85,B 0,C 180,E1 -5992.036,E2 -5992.036} C_VEL
LIN {X 0,Y 495.36,Z 740.049,A -85,B 0,C 180,E1 -5992.626,E2 -5992.626} C_VEL
LIN {X 0,Y 495.602,Z 732.35,A -85,B 0,C 180,E1 -5993.931,E2 -5993.931} C_VEL
LIN {X 0,Y 495.945,Z 723.645,A -85,B 0,C 180,E1 -5995.117,E2 -5995.117} C_VEL
LIN {X 0,Y 496.294,Z 714.665,A -85,B 0,C 180,E1 -5996.111,E2 -5996.111} C_VEL
LIN {X 0,Y 496.687,Z 703.401,A -85,B 0,C 180,E1 -5997.112,E2 -5997.112} C_VEL
LIN {X 0,Y 497.063,Z 691.609,A -85,B 0,C 180,E1 -5997.943,E2 -5997.943} C_VEL
LIN {X 0,Y 497.445,Z 679.283,A -85,B 0,C 180,E1 -5998.602,E2 -5998.602} C_VEL
LIN {X 0,Y 497.595,Z 668.006,A -85,B 0,C 180,E1 -5999.056,E2 -5999.056} C_VEL
LIN {X 0,Y 495.496,Z 656.529,A -85,B 0,C 180,E1 -5999.447,E2 -5999.447} C_VEL
LIN {X 0,Y 495.045,Z 654.252,A -85,B 0,C 180,E1 -5999.517,E2 -5999.517} C_VEL
LIN {X 0,Y 495.115,Z 650.14,A -85,B 0,C 180,E1 -6002.068,E2 -6002.068} C_VEL
LIN {X 0,Y 495.137,Z 645.805,A -85,B 0,C 180,E1 -6004.797,E2 -6004.797} C_VEL
LIN {X 0,Y 495.249,Z 641.605,A -85,B 0,C 180,E1 -6007.471,E2 -6007.471} C_VEL
LIN {X 0,Y 495.361,Z 637.523,A -85,B 0,C 180,E1 -6010.092,E2 -6010.092} C_VEL
LIN {X 0,Y 495.423,Z 633.596,A -85,B 0,C 180,E1 -6012.668,E2 -6012.668} C_VEL
LIN {X 0,Y 495.55,Z 629.762,A -85,B 0,C 180,E1 -6015.21,E2 -6015.21} C_VEL
LIN {X 0,Y 495.694,Z 624.833,A -85,B 0,C 180,E1 -6018.551,E2 -6018.551} C_VEL
LIN {X 0,Y 495.68,Z 622.743,A -85,B 0,C 180,E1 -6020.204,E2 -6020.204} C_VEL
LIN {X 0,Y 495.897,Z 622.717,A -85,B 0,C 180,E1 -6022.777,E2 -6022.777} C_VEL
LIN {X 0,Y 495.843,Z 622.723,A -85,B 0,C 180,E1 -6025.121,E2 -6025.121} C_VEL
LIN {X 0,Y 495.998,Z 622.701,A -85,B 0,C 180,E1 -6027.563,E2 -6027.563} C_VEL
LIN {X 0,Y 496.003,Z 622.702,A -85,B 0,C 180,E1 -6030,E2 -6030} C_VEL
LIN {X 0,Y 495.997,Z 622.703,A -85,B 0,C 180,E1 -6032.436,E2 -6032.436} C_VEL
LIN {X 0,Y 495.893,Z 622.715,A -85,B 0,C 180,E1 -6035.693,E2 -6035.693} C_VEL
LIN {X 0,Y 495.823,Z 622.725,A -85,B 0,C 180,E1 -6038.148,E2 -6038.148} C_VEL
LIN {X 0,Y 495.466,Z 622.795,A -85,B 0,C 180,E1 -6040.936,E2 -6040.936} C_VEL
LIN {X 0,Y 495.335,Z 627.955,A -85,B 0,C 180,E1 -6043.957,E2 -6043.957} C_VEL
LIN {X 0,Y 495.285,Z 632.255,A -85,B 0,C 180,E1 -6046.486,E2 -6046.486} C_VEL
LIN {X 0,Y 495.215,Z 636.565,A -85,B 0,C 180,E1 -6049.051,E2 -6049.051} C_VEL
LIN {X 0,Y 495.149,Z 640.932,A -85,B 0,C 180,E1 -6051.656,E2 -6051.656} C_VEL
LIN {X 0,Y 495.112,Z 646.018,A -85,B 0,C 180,E1 -6054.705,E2 -6054.705} C_VEL
LIN {X 0,Y 495.033,Z 651.385,A -85,B 0,C 180,E1 -6057.937,E2 -6057.937} C_VEL
LIN {X 0,Y 495.029,Z 654.233,A -85,B 0,C 180,E1 -6059.59,E2 -6059.59} C_VEL
LIN {X 0,Y 497.251,Z 665.706,A -85,B 0,C 180,E1 -6059.956,E2 -6059.956} C_VEL
LIN {X 0,Y 497.711,Z 671.09,A -85,B 0,C 180,E1 -6060.153,E2 -6060.153} C_VEL
LIN {X 0,Y 497.293,Z 683.442,A -85,B 0,C 180,E1 -6060.699,E2 -6060.699} C_VEL
LIN {X 0,Y 496.977,Z 693.999,A -85,B 0,C 180,E1 -6061.312,E2 -6061.312} C_VEL
LIN {X 0,Y 496.623,Z 703.398,A -85,B 0,C 180,E1 -6061.986,E2 -6061.986} C_VEL
LIN {X 0,Y 496.309,Z 712.651,A -85,B 0,C 180,E1 -6062.795,E2 -6062.795} C_VEL
LIN {X 0,Y 495.979,Z 722.052,A -85,B 0,C 180,E1 -6063.791,E2 -6063.791} C_VEL
LIN {X 0,Y 495.595,Z 731.806,A -85,B 0,C 180,E1 -6065.084,E2 -6065.084} C_VEL
LIN {X 0,Y 495.374,Z 738.949,A -85,B 0,C 180,E1 -6066.275,E2 -6066.275} C_VEL
LIN {X 0,Y 495.218,Z 744.315,A -85,B 0,C 180,E1 -6067.369,E2 -6067.369} C_VEL
LIN {X 0,Y 495.159,Z 747.5,A -85,B 0,C 180,E1 -6068.127,E2 -6068.127} C_VEL
LIN {X 0,Y 495.058,Z 751.104,A -85,B 0,C 180,E1 -6069.177,E2 -6069.177} C_VEL
LIN {X 0,Y 494.902,Z 755.084,A -85,B 0,C 180,E1 -6070.785,E2 -6070.785} C_VEL
LIN {X 0,Y 494.909,Z 756.879,A -85,B 0,C 180,E1 -6071.868,E2 -6071.868} C_VEL
LIN {X 0,Y 494.907,Z 757.97,A -85,B 0,C 180,E1 -6072.97,E2 -6072.97} C_VEL
LIN {X 0,Y 494.921,Z 758.324,A -85,B 0,C 180,E1 -6074.091,E2 -6074.091} C_VEL
LIN {X 0,Y 494.921,Z 757.906,A -85,B 0,C 180,E1 -6075.235,E2 -6075.235} C_VEL
LIN {X 0,Y 494.896,Z 756.663,A -85,B 0,C 180,E1 -6076.406,E2 -6076.406} C_VEL
LIN {X 0,Y 494.984,Z 754.555,A -85,B 0,C 180,E1 -6077.588,E2 -6077.588} C_VEL
LIN {X 0,Y 495.091,Z 751.473,A -85,B 0,C 180,E1 -6078.794,E2 -6078.794} C_VEL
LIN {X 0,Y 495.183,Z 746.123,A -85,B 0,C 180,E1 -6080.307,E2 -6080.307} C_VEL
LIN {X 0,Y 495.344,Z 741.311,A -85,B 0,C 180,E1 -6081.371,E2 -6081.371} C_VEL
LIN {X 0,Y 495.528,Z 734.526,A -85,B 0,C 180,E1 -6082.583,E2 -6082.583} C_VEL
LIN {X 0,Y 495.817,Z 726.789,A -85,B 0,C 180,E1 -6083.708,E2 -6083.708} C_VEL
LIN {X 0,Y 496.125,Z 718.623,A -85,B 0,C 180,E1 -6084.689,E2 -6084.689} C_VEL
LIN {X 0,Y 496.515,Z 707.671,A -85,B 0,C 180,E1 -6085.761,E2 -6085.761} C_VEL
LIN {X 0,Y 496.942,Z 696.23,A -85,B 0,C 180,E1 -6086.636,E2 -6086.636} C_VEL
LIN {X 0,Y 497.244,Z 685.717,A -85,B 0,C 180,E1 -6087.274,E2 -6087.274} C_VEL
LIN {X 0,Y 497.579,Z 675.64,A -85,B 0,C 180,E1 -6087.754,E2 -6087.754} C_VEL
LIN {X 0,Y 497.528,Z 667.704,A -85,B 0,C 180,E1 -6088.064,E2 -6088.064} C_VEL
LIN {X 0,Y 495.264,Z 655.484,A -85,B 0,C 180,E1 -6088.468,E2 -6088.468} C_VEL
LIN {X 0,Y 495.041,Z 654.213,A -85,B 0,C 180,E1 -6088.512,E2 -6088.512} C_VEL
LIN {X 0,Y 495.091,Z 648.966,A -85,B 0,C 180,E1 -6091.655,E2 -6091.655} C_VEL
LIN {X 0,Y 495.141,Z 645.195,A -85,B 0,C 180,E1 -6093.895,E2 -6093.895} C_VEL
LIN {X 0,Y 495.147,Z 640.566,A -85,B 0,C 180,E1 -6096.583,E2 -6096.583} C_VEL
LIN {X 0,Y 495.231,Z 635.55,A -85,B 0,C 180,E1 -6099.491,E2 -6099.491} C_VEL
LIN {X 0,Y 495.274,Z 630.078,A -85,B 0,C 180,E1 -6102.663,E2 -6102.663} C_VEL
LIN {X 0,Y 495.351,Z 625.469,A -85,B 0,C 180,E1 -6105.204,E2 -6105.204} C_VEL
LIN {X 0,Y 495.348,Z 622.787,A -85,B 0,C 180,E1 -6106.67,E2 -6106.67} C_VEL
LIN {X 0,Y 495.698,Z 622.743,A -85,B 0,C 180,E1 -6108.551,E2 -6108.551} C_VEL
LIN {X 0,Y 495.87,Z 622.721,A -85,B 0,C 180,E1 -6111.852,E2 -6111.852} C_VEL
LIN {X 0,Y 495.895,Z 622.718,A -85,B 0,C 180,E1 -6114.306,E2 -6114.306} C_VEL
LIN {X 0,Y 495.991,Z 622.704,A -85,B 0,C 180,E1 -6117.564,E2 -6117.564} C_VEL
LIN {X 0,Y 495.994,Z 622.704,A -85,B 0,C 180,E1 -6120,E2 -6120} C_VEL
LIN {X 0,Y 495.99,Z 622.706,A -85,B 0,C 180,E1 -6122.436,E2 -6122.436} C_VEL
LIN {X 0,Y 495.894,Z 622.716,A -85,B 0,C 180,E1 -6125.693,E2 -6125.693} C_VEL
LIN {X 0,Y 495.87,Z 622.719,A -85,B 0,C 180,E1 -6128.148,E2 -6128.148} C_VEL
LIN {X 0,Y 495.851,Z 622.722,A -85,B 0,C 180,E1 -6131.445,E2 -6131.445} C_VEL
LIN {X 0,Y 495.787,Z 622.731,A -85,B 0,C 180,E1 -6134.783,E2 -6134.783} C_VEL
LIN {X 0,Y 495.784,Z 622.73,A -85,B 0,C 180,E1 -6137.319,E2 -6137.319} C_VEL
LIN {X 0,Y 495.775,Z 622.733,A -85,B 0,C 180,E1 -6139.89,E2 -6139.89} C_VEL
LIN {X 0,Y 495.755,Z 622.735,A -85,B 0,C 180,E1 -6142.861,E2 -6142.861} C_VEL
LIN {X 0,Y 495.797,Z 622.729,A -85,B 0,C 180,E1 -6146.068,E2 -6146.068} C_VEL
LIN {X 0,Y 495.778,Z 622.73,A -85,B 0,C 180,E1 -6148.815,E2 -6148.815} C_VEL
LIN {X 0,Y 495.757,Z 622.733,A -85,B 0,C 180,E1 -6151.727,E2 -6151.727} C_VEL
LIN {X 0,Y 495.772,Z 622.731,A -85,B 0,C 180,E1 -6154.695,E2 -6154.695} C_VEL
LIN {X 0,Y 495.729,Z 622.736,A -85,B 0,C 180,E1 -6157.562,E2 -6157.562} C_VEL
LIN {X 0,Y 495.764,Z 622.733,A -85,B 0,C 180,E1 -6160.7,E2 -6160.7} C_VEL
LIN {X 0,Y 495.732,Z 622.736,A -85,B 0,C 180,E1 -6164.001,E2 -6164.001} C_VEL
LIN {X 0,Y 495.724,Z 622.737,A -85,B 0,C 180,E1 -6167.118,E2 -6167.118} C_VEL
LIN {X 0,Y 495.757,Z 622.734,A -85,B 0,C 180,E1 -6169.953,E2 -6169.953} C_VEL
LIN {X 0,Y 495.785,Z 622.836,A -85,B 0,C 180,E1 -6171.672,E2 -6171.672} C_VEL
LIN {X 0,Y 496.511,Z 627.258,A -85,B 0,C 180,E1 -6173.787,E2 -6173.787} C_VEL
LIN {X 0,Y 496.515,Z 632.176,A -85,B 0,C 180,E1 -6176.006,E2 -6176.006} C_VEL
LIN {X 0,Y 496.231,Z 638.785,A -85,B 0,C 180,E1 -6178.873,E2 -6178.873} C_VEL
LIN {X 0,Y 496.058,Z 644.899,A -85,B 0,C 180,E1 -6181.45,E2 -6181.45} C_VEL
LIN {X 0,Y 495.85,Z 652.09,A -85,B 0,C 180,E1 -6184.387,E2 -6184.387} C_VEL
LIN {X 0,Y 495.65,Z 659.922,A -85,B 0,C 180,E1 -6187.491,E2 -6187.491} C_VEL
LIN {X 0,Y 495.533,Z 666.626,A -85,B 0,C 180,E1 -6190.1,E2 -6190.1} C_VEL
LIN {X 0,Y 495.352,Z 675.599,A -85,B 0,C 180,E1 -6193.516,E2 -6193.516} C_VEL
LIN {X 0,Y 495.273,Z 680.974,A -85,B 0,C 180,E1 -6195.504,E2 -6195.504} C_VEL
LIN {X 0,Y 497.518,Z 694.556,A -85,B 0,C 180,E1 -6195.91,E2 -6195.91} C_VEL
LIN {X 0,Y 497.576,Z 702.746,A -85,B 0,C 180,E1 -6196.211,E2 -6196.211} C_VEL
LIN {X 0,Y 497.198,Z 713.792,A -85,B 0,C 180,E1 -6196.721,E2 -6196.721} C_VEL
LIN {X 0,Y 496.846,Z 725.525,A -85,B 0,C 180,E1 -6197.428,E2 -6197.428} C_VEL
LIN {X 0,Y 496.546,Z 736.331,A -85,B 0,C 180,E1 -6198.261,E2 -6198.261} C_VEL
LIN {X 0,Y 496.127,Z 746.06,A -85,B 0,C 180,E1 -6199.182,E2 -6199.182} C_VEL
LIN {X 0,Y 495.813,Z 754.926,A -85,B 0,C 180,E1 -6200.207,E2 -6200.207} C_VEL
LIN {X 0,Y 495.526,Z 763.574,A -85,B 0,C 180,E1 -6201.436,E2 -6201.436} C_VEL
LIN {X 0,Y 495.274,Z 770.482,A -85,B 0,C 180,E1 -6202.663,E2 -6202.663} C_VEL
LIN {X 0,Y 495.164,Z 776.504,A -85,B 0,C 180,E1 -6204.012,E2 -6204.012} C_VEL
LIN {X 0,Y 495.039,Z 780.36,A -85,B 0,C 180,E1 -6205.114,E2 -6205.114} C_VEL
LIN {X 0,Y 495.046,Z 782.659,A -85,B 0,C 180,E1 -6205.93,E2 -6205.93} C_VEL
LIN {X 0,Y 495.043,Z 784.522,A -85,B 0,C 180,E1 -6206.745,E2 -6206.745} C_VEL
LIN {X 0,Y 494.961,Z 786.913,A -85,B 0,C 180,E1 -6208.373,E2 -6208.373} C_VEL
LIN {X 0,Y 494.898,Z 787.734,A -85,B 0,C 180,E1 -6210,E2 -6210} C_VEL
LIN {X 0,Y 494.961,Z 786.91,A -85,B 0,C 180,E1 -6211.628,E2 -6211.628} C_VEL
LIN {X 0,Y 495.043,Z 784.516,A -85,B 0,C 180,E1 -6213.256,E2 -6213.256} C_VEL
LIN {X 0,Y 495.027,Z 781.573,A -85,B 0,C 180,E1 -6214.479,E2 -6214.479} C_VEL
LIN {X 0,Y 495.174,Z 777.593,A -85,B 0,C 180,E1 -6215.702,E2 -6215.702} C_VEL
LIN {X 0,Y 495.251,Z 771.568,A -85,B 0,C 180,E1 -6217.113,E2 -6217.113} C_VEL
LIN {X 0,Y 495.473,Z 764.773,A -85,B 0,C 180,E1 -6218.36,E2 -6218.36} C_VEL
LIN {X 0,Y 495.747,Z 756.466,A -85,B 0,C 180,E1 -6219.589,E2 -6219.589} C_VEL
LIN {X 0,Y 496.04,Z 747.947,A -85,B 0,C 180,E1 -6220.614,E2 -6220.614} C_VEL
LIN {X 0,Y 496.504,Z 737.427,A -85,B 0,C 180,E1 -6221.637,E2 -6221.637} C_VEL
LIN {X 0,Y 496.829,Z 725.569,A -85,B 0,C 180,E1 -6222.563,E2 -6222.563} C_VEL
LIN {X 0,Y 497.191,Z 713.664,A -85,B 0,C 180,E1 -6223.28,E2 -6223.28} C_VEL
LIN {X 0,Y 497.569,Z 701.284,A -85,B 0,C 180,E1 -6223.842,E2 -6223.842} C_VEL
LIN {X 0,Y 497.485,Z 694.4,A -85,B 0,C 180,E1 -6224.092,E2 -6224.092} C_VEL
LIN {X 0,Y 495.268,Z 680.775,A -85,B 0,C 180,E1 -6224.51,E2 -6224.51} C_VEL
LIN {X 0,Y 495.376,Z 673.23,A -85,B 0,C 180,E1 -6227.334,E2 -6227.334} C_VEL
LIN {X 0,Y 495.572,Z 664.54,A -85,B 0,C 180,E1 -6230.612,E2 -6230.612} C_VEL
LIN {X 0,Y 495.67,Z 656.224,A -85,B 0,C 180,E1 -6233.835,E2 -6233.835} C_VEL
LIN {X 0,Y 495.88,Z 648.923,A -85,B 0,C 180,E1 -6236.762,E2 -6236.762} C_VEL
LIN {X 0,Y 496.095,Z 641.772,A -85,B 0,C 180,E1 -6239.725,E2 -6239.725} C_VEL
LIN {X 0,Y 496.354,Z 635.212,A -85,B 0,C 180,E1 -6242.551,E2 -6242.551} C_VEL
LIN {X 0,Y 496.589,Z 628.755,A -85,B 0,C 180,E1 -6245.469,E2 -6245.469} C_VEL
LIN {X 0,Y 495.929,Z 623.51,A -85,B 0,C 180,E1 -6248.058,E2 -6248.058} C_VEL
LIN {X 0,Y 495.757,Z 622.731,A -85,B 0,C 180,E1 -6248.591,E2 -6248.591} C_VEL
LIN {X 0,Y 495.78,Z 622.732,A -85,B 0,C 180,E1 -6251.779,E2 -6251.779} C_VEL
LIN {X 0,Y 495.751,Z 622.735,A -85,B 0,C 180,E1 -6255.139,E2 -6255.139} C_VEL
LIN {X 0,Y 495.758,Z 622.735,A -85,B 0,C 180,E1 -6258.219,E2 -6258.219} C_VEL
LIN {X 0,Y 495.752,Z 622.736,A -85,B 0,C 180,E1 -6261.408,E2 -6261.408} C_VEL
LIN {X 0,Y 495.753,Z 622.735,A -85,B 0,C 180,E1 -6264.463,E2 -6264.463} C_VEL
LIN {X 0,Y 495.77,Z 622.733,A -85,B 0,C 180,E1 -6267.406,E2 -6267.406} C_VEL
LIN {X 0,Y 495.768,Z 622.732,A -85,B 0,C 180,E1 -6270.254,E2 -6270.254} C_VEL
LIN {X 0,Y 495.825,Z 622.726,A -85,B 0,C 180,E1 -6273.251,E2 -6273.251} C_VEL
LIN {X 0,Y 495.754,Z 622.733,A -85,B 0,C 180,E1 -6275.725,E2 -6275.725} C_VEL
LIN {X 0,Y 495.744,Z 622.736,A -85,B 0,C 180,E1 -6278.371,E2 -6278.371} C_VEL
LIN {X 0,Y 495.786,Z 622.73,A -85,B 0,C 180,E1 -6280.972,E2 -6280.972} C_VEL
LIN {X 0,Y 495.781,Z 622.732,A -85,B 0,C 180,E1 -6283.53,E2 -6283.53} C_VEL
LIN {X 0,Y 495.796,Z 622.728,A -85,B 0,C 180,E1 -6286.056,E2 -6286.056} C_VEL
LIN {X 0,Y 495.853,Z 622.723,A -85,B 0,C 180,E1 -6288.555,E2 -6288.555} C_VEL
LIN {X 0,Y 495.875,Z 622.718,A -85,B 0,C 180,E1 -6291.852,E2 -6291.852} C_VEL
LIN {X 0,Y 495.897,Z 622.715,A -85,B 0,C 180,E1 -6294.307,E2 -6294.307} C_VEL
LIN {X 0,Y 495.994,Z 622.704,A -85,B 0,C 180,E1 -6297.564,E2 -6297.564} C_VEL
LIN {X 0,Y 495.999,Z 622.704,A -85,B 0,C 180,E1 -6300,E2 -6300} C_VEL
LIN {X 0,Y 495.996,Z 622.705,A -85,B 0,C 180,E1 -6302.436,E2 -6302.436} C_VEL
LIN {X 0,Y 495.899,Z 622.717,A -85,B 0,C 180,E1 -6305.693,E2 -6305.693} C_VEL
LIN {X 0,Y 495.868,Z 622.721,A -85,B 0,C 180,E1 -6308.148,E2 -6308.148} C_VEL
LIN {X 0,Y 495.733,Z 622.949,A -85,B 0,C 180,E1 -6309.795,E2 -6309.795} C_VEL
LIN {X 0,Y 495.66,Z 626.47,A -85,B 0,C 180,E1 -6312.28,E2 -6312.28} C_VEL
LIN {X 0,Y 495.543,Z 631.349,A -85,B 0,C 180,E1 -6315.633,E2 -6315.633} C_VEL
LIN {X 0,Y 495.441,Z 635.136,A -85,B 0,C 180,E1 -6318.185,E2 -6318.185} C_VEL
LIN {X 0,Y 495.351,Z 639.045,A -85,B 0,C 180,E1 -6320.775,E2 -6320.775} C_VEL
LIN {X 0,Y 495.222,Z 643.107,A -85,B 0,C 180,E1 -6323.414,E2 -6323.414} C_VEL
LIN {X 0,Y 495.196,Z 648.056,A -85,B 0,C 180,E1 -6326.604,E2 -6326.604} C_VEL
LIN {X 0,Y 495.083,Z 653.111,A -85,B 0,C 180,E1 -6329.792,E2 -6329.792} C_VEL
LIN {X 0,Y 495.054,Z 654.365,A -85,B 0,C 180,E1 -6330.57,E2 -6330.57} C_VEL
LIN {X 0,Y 497.607,Z 668.013,A -85,B 0,C 180,E1 -6331.032,E2 -6331.032} C_VEL
LIN {X 0,Y 497.452,Z 679.953,A -85,B 0,C 180,E1 -6331.516,E2 -6331.516} C_VEL
LIN {X 0,Y 497.096,Z 690.88,A -85,B 0,C 180,E1 -6332.1,E2 -6332.1} C_VEL
LIN {X 0,Y 496.759,Z 702.26,A -85,B 0,C 180,E1 -6332.883,E2 -6332.883} C_VEL
LIN {X 0,Y 496.31,Z 712.52,A -85,B 0,C 180,E1 -6333.766,E2 -6333.766} C_VEL
LIN {X 0,Y 496.001,Z 722.933,A -85,B 0,C 180,E1 -6334.881,E2 -6334.881} C_VEL
LIN {X 0,Y 495.633,Z 731.829,A -85,B 0,C 180,E1 -6336.074,E2 -6336.074} C_VEL
LIN {X 0,Y 495.36,Z 739.686,A -85,B 0,C 180,E1 -6337.391,E2 -6337.391} C_VEL
LIN {X 0,Y 495.205,Z 745.807,A -85,B 0,C 180,E1 -6338.687,E2 -6338.687} C_VEL
LIN {X 0,Y 495.065,Z 750.447,A -85,B 0,C 180,E1 -6339.951,E2 -6339.951} C_VEL
LIN {X 0,Y 495.043,Z 753.904,A -85,B 0,C 180,E1 -6341.199,E2 -6341.199} C_VEL
LIN {X 0,Y 494.965,Z 756.283,A -85,B 0,C 180,E1 -6342.409,E2 -6342.409} C_VEL
LIN {X 0,Y 494.896,Z 758.062,A -85,B 0,C 180,E1 -6344.095,E2 -6344.095} C_VEL
LIN {X 0,Y 494.925,Z 758.321,A -85,B 0,C 180,E1 -6345.236,E2 -6345.236} C_VEL
LIN {X 0,Y 494.898,Z 757.796,A -85,B 0,C 180,E1 -6346.406,E2 -6346.406} C_VEL
LIN {X 0,Y 494.953,Z 756.403,A -85,B 0,C 180,E1 -6347.593,E2 -6347.593} C_VEL
LIN {X 0,Y 495.021,Z 753.042,A -85,B 0,C 180,E1 -6349.226,E2 -6349.226} C_VEL
LIN {X 0,Y 495.095,Z 749.897,A -85,B 0,C 180,E1 -6350.298,E2 -6350.298} C_VEL
LIN {X 0,Y 495.237,Z 744.829,A -85,B 0,C 180,E1 -6351.621,E2 -6351.621} C_VEL
LIN {X 0,Y 495.36,Z 740.049,A -85,B 0,C 180,E1 -6352.626,E2 -6352.626} C_VEL
LIN {X 0,Y 494.811,Z 736.961,A -85,B 0,C 180,E1 -6353.201,E2 -6353.201} C_VEL
LIN {X 0,Y 492.171,Z 731.592,A -85,B 0,C 180,E1 -6354.123,E2 -6354.123} C_VEL
LIN {X 0,Y 489.553,Z 725.724,A -85,B 0,C 180,E1 -6355.005,E2 -6355.005} C_VEL
LIN {X 0,Y 489.04,Z 721.727,A -85,B 0,C 180,E1 -6355.512,E2 -6355.512} C_VEL
LIN {X 0,Y 489.393,Z 712.02,A -85,B 0,C 180,E1 -6356.546,E2 -6356.546} C_VEL
LIN {X 0,Y 489.835,Z 701.914,A -85,B 0,C 180,E1 -6357.418,E2 -6357.418} C_VEL
LIN {X 0,Y 490.169,Z 690.524,A -85,B 0,C 180,E1 -6358.202,E2 -6358.202} C_VEL
LIN {X 0,Y 490.598,Z 678.57,A -85,B 0,C 180,E1 -6358.835,E2 -6358.835} C_VEL
LIN {X 0,Y 490.709,Z 669.03,A -85,B 0,C 180,E1 -6359.225,E2 -6359.225} C_VEL
LIN {X 0,Y 488.544,Z 657.365,A -85,B 0,C 180,E1 -6359.639,E2 -6359.639} C_VEL
LIN {X 0,Y 487.972,Z 654.455,A -85,B 0,C 180,E1 -6359.729,E2 -6359.729} C_VEL
LIN {X 0,Y 488.026,Z 649.942,A -85,B 0,C 180,E1 -6362.559,E2 -6362.559} C_VEL
LIN {X 0,Y 488.082,Z 645.599,A -85,B 0,C 180,E1 -6365.318,E2 -6365.318} C_VEL
LIN {X 0,Y 488.171,Z 641.408,A -85,B 0,C 180,E1 -6368.018,E2 -6368.018} C_VEL
LIN {X 0,Y 488.276,Z 637.361,A -85,B 0,C 180,E1 -6370.667,E2 -6370.667} C_VEL
LIN {X 0,Y 488.376,Z 633.443,A -85,B 0,C 180,E1 -6373.273,E2 -6373.273} C_VEL
LIN {X 0,Y 488.467,Z 629.635,A -85,B 0,C 180,E1 -6375.842,E2 -6375.842} C_VEL
LIN {X 0,Y 488.635,Z 625.908,A -85,B 0,C 180,E1 -6378.383,E2 -6378.383} C_VEL
LIN {X 0,Y 488.605,Z 623.625,A -85,B 0,C 180,E1 -6380.06,E2 -6380.06} C_VEL
LIN {X 0,Y 488.87,Z 623.593,A -85,B 0,C 180,E1 -6382.725,E2 -6382.725} C_VEL
LIN {X 0,Y 488.813,Z 623.599,A -85,B 0,C 180,E1 -6385.051,E2 -6385.051} C_VEL
LIN {X 0,Y 488.965,Z 623.577,A -85,B 0,C 180,E1 -6387.528,E2 -6387.528} C_VEL
LIN {X 0,Y 488.959,Z 623.582,A -85,B 0,C 180,E1 -6390.823,E2 -6390.823} C_VEL
LIN {X 0,Y 488.965,Z 623.579,A -85,B 0,C 180,E1 -6392.471,E2 -6392.471} C_VEL
LIN {X 0,Y 488.851,Z 623.592,A -85,B 0,C 180,E1 -6395.775,E2 -6395.775} C_VEL
LIN {X 0,Y 488.758,Z 623.605,A -85,B 0,C 180,E1 -6398.267,E2 -6398.267} C_VEL
LIN {X 0,Y 488.407,Z 623.77,A -85,B 0,C 180,E1 -6401.096,E2 -6401.096} C_VEL
LIN {X 0,Y 488.265,Z 628.974,A -85,B 0,C 180,E1 -6404.163,E2 -6404.163} C_VEL
LIN {X 0,Y 488.203,Z 633.292,A -85,B 0,C 180,E1 -6406.733,E2 -6406.733} C_VEL
LIN {X 0,Y 488.143,Z 637.655,A -85,B 0,C 180,E1 -6409.338,E2 -6409.338} C_VEL
LIN {X 0,Y 488.06,Z 642.062,A -85,B 0,C 180,E1 -6411.987,E2 -6411.987} C_VEL
LIN {X 0,Y 488.038,Z 646.85,A -85,B 0,C 180,E1 -6414.874,E2 -6414.874} C_VEL
LIN {X 0,Y 487.95,Z 651.106,A -85,B 0,C 180,E1 -6417.445,E2 -6417.445} C_VEL
LIN {X 0,Y 487.991,Z 654.349,A -85,B 0,C 180,E1 -6419.377,E2 -6419.377} C_VEL
LIN {X 0,Y 490.245,Z 666.087,A -85,B 0,C 180,E1 -6419.76,E2 -6419.76} C_VEL
LIN {X 0,Y 490.806,Z 671.294,A -85,B 0,C 180,E1 -6419.959,E2 -6419.959} C_VEL
LIN {X 0,Y 490.395,Z 683.533,A -85,B 0,C 180,E1 -6420.505,E2 -6420.505} C_VEL
LIN {X 0,Y 490.082,Z 693.421,A -85,B 0,C 180,E1 -6421.081,E2 -6421.081} C_VEL
LIN {X 0,Y 489.673,Z 703.799,A -85,B 0,C 180,E1 -6421.833,E2 -6421.833} C_VEL
LIN {X 0,Y 489.31,Z 713.626,A -85,B 0,C 180,E1 -6422.711,E2 -6422.711} C_VEL
LIN {X 0,Y 488.923,Z 723.367,A -85,B 0,C 180,E1 -6423.781,E2 -6423.781} C_VEL
LIN {X 0,Y 488.585,Z 731.782,A -85,B 0,C 180,E1 -6424.924,E2 -6424.924} C_VEL
LIN {X 0,Y 488.328,Z 739.128,A -85,B 0,C 180,E1 -6426.161,E2 -6426.161} C_VEL
LIN {X 0,Y 488.155,Z 744.216,A -85,B 0,C 180,E1 -6427.205,E2 -6427.205} C_VEL
LIN {X 0,Y 488.071,Z 748.445,A -85,B 0,C 180,E1 -6428.256,E2 -6428.256} C_VEL
LIN {X 0,Y 487.948,Z 751.929,A -85,B 0,C 180,E1 -6429.326,E2 -6429.326} C_VEL
LIN {X 0,Y 487.848,Z 754.648,A -85,B 0,C 180,E1 -6430.411,E2 -6430.411} C_VEL
LIN {X 0,Y 487.816,Z 756.65,A -85,B 0,C 180,E1 -6431.507,E2 -6431.507} C_VEL
LIN {X 0,Y 487.828,Z 758.006,A -85,B 0,C 180,E1 -6432.714,E2 -6432.714} C_VEL
LIN {X 0,Y 487.826,Z 758.506,A -85,B 0,C 180,E1 -6433.917,E2 -6433.917} C_VEL
LIN {X 0,Y 487.838,Z 758.189,A -85,B 0,C 180,E1 -6435.096,E2 -6435.096} C_VEL
LIN {X 0,Y 487.795,Z 757.106,A -85,B 0,C 180,E1 -6436.245,E2 -6436.245} C_VEL
LIN {X 0,Y 487.917,Z 754.051,A -85,B 0,C 180,E1 -6437.949,E2 -6437.949} C_VEL
LIN {X 0,Y 488.01,Z 751.082,A -85,B 0,C 180,E1 -6439.06,E2 -6439.06} C_VEL
LIN {X 0,Y 488.123,Z 746.073,A -85,B 0,C 180,E1 -6440.457,E2 -6440.457} C_VEL
LIN {X 0,Y 488.33,Z 740.003,A -85,B 0,C 180,E1 -6441.767,E2 -6441.767} C_VEL
LIN {X 0,Y 488.533,Z 733.961,A -85,B 0,C 180,E1 -6442.828,E2 -6442.828} C_VEL
LIN {X 0,Y 488.796,Z 726.763,A -85,B 0,C 180,E1 -6443.878,E2 -6443.878} C_VEL
LIN {X 0,Y 489.176,Z 717.605,A -85,B 0,C 180,E1 -6444.976,E2 -6444.976} C_VEL
LIN {X 0,Y 489.603,Z 706.213,A -85,B 0,C 180,E1 -6446.065,E2 -6446.065} C_VEL
LIN {X 0,Y 490.026,Z 695.648,A -85,B 0,C 180,E1 -6446.866,E2 -6446.866} C_VEL
LIN {X 0,Y 490.413,Z 684.329,A -85,B 0,C 180,E1 -6447.545,E2 -6447.545} C_VEL
LIN {X 0,Y 490.782,Z 672.536,A -85,B 0,C 180,E1 -6448.086,E2 -6448.086} C_VEL
LIN {X 0,Y 490.554,Z 668.332,A -85,B 0,C 180,E1 -6448.251,E2 -6448.251} C_VEL
LIN {X 0,Y 488.296,Z 656.157,A -85,B 0,C 180,E1 -6448.666,E2 -6448.666} C_VEL
LIN {X 0,Y 487.989,Z 654.408,A -85,B 0,C 180,E1 -6448.72,E2 -6448.72} C_VEL
LIN {X 0,Y 488.01,Z 649.566,A -85,B 0,C 180,E1 -6451.625,E2 -6451.625} C_VEL
LIN {X 0,Y 488.041,Z 644.92,A -85,B 0,C 180,E1 -6454.405,E2 -6454.405} C_VEL
LIN {X 0,Y 488.09,Z 640.208,A -85,B 0,C 180,E1 -6457.15,E2 -6457.15} C_VEL
LIN {X 0,Y 488.178,Z 635.778,A -85,B 0,C 180,E1 -6459.787,E2 -6459.787} C_VEL
LIN {X 0,Y 488.22,Z 631.173,A -85,B 0,C 180,E1 -6462.404,E2 -6462.404} C_VEL
LIN {X 0,Y 488.28,Z 626.568,A -85,B 0,C 180,E1 -6464.984,E2 -6464.984} C_VEL
LIN {X 0,Y 488.287,Z 623.667,A -85,B 0,C 180,E1 -6466.686,E2 -6466.686} C_VEL
LIN {X 0,Y 488.624,Z 623.624,A -85,B 0,C 180,E1 -6468.383,E2 -6468.383} C_VEL
LIN {X 0,Y 488.776,Z 623.605,A -85,B 0,C 180,E1 -6470.899,E2 -6470.899} C_VEL
LIN {X 0,Y 488.83,Z 623.598,A -85,B 0,C 180,E1 -6473.395,E2 -6473.395} C_VEL
LIN {X 0,Y 488.701,Z 623.613,A -85,B 0,C 180,E1 -6475.877,E2 -6475.877} C_VEL
LIN {X 0,Y 488.959,Z 623.58,A -85,B 0,C 180,E1 -6477.529,E2 -6477.529} C_VEL
LIN {X 0,Y 488.965,Z 623.58,A -85,B 0,C 180,E1 -6480,E2 -6480} C_VEL
LIN {X 0,Y 488.958,Z 623.582,A -85,B 0,C 180,E1 -6482.471,E2 -6482.471} C_VEL
LIN {X 0,Y 488.853,Z 623.593,A -85,B 0,C 180,E1 -6485.776,E2 -6485.776} C_VEL
LIN {X 0,Y 488.815,Z 623.598,A -85,B 0,C 180,E1 -6488.266,E2 -6488.266} C_VEL
LIN {X 0,Y 488.804,Z 623.6,A -85,B 0,C 180,E1 -6491.612,E2 -6491.612} C_VEL
LIN {X 0,Y 488.758,Z 623.605,A -85,B 0,C 180,E1 -6495.001,E2 -6495.001} C_VEL
LIN {X 0,Y 488.751,Z 623.606,A -85,B 0,C 180,E1 -6498.442,E2 -6498.442} C_VEL
LIN {X 0,Y 488.704,Z 623.611,A -85,B 0,C 180,E1 -6501.071,E2 -6501.071} C_VEL
LIN {X 0,Y 488.691,Z 623.613,A -85,B 0,C 180,E1 -6503.746,E2 -6503.746} C_VEL
LIN {X 0,Y 488.796,Z 623.601,A -85,B 0,C 180,E1 -6506.946,E2 -6506.946} C_VEL
LIN {X 0,Y 488.716,Z 623.61,A -85,B 0,C 180,E1 -6510.365,E2 -6510.365} C_VEL
LIN {X 0,Y 488.733,Z 623.608,A -85,B 0,C 180,E1 -6513.485,E2 -6513.485} C_VEL
LIN {X 0,Y 488.685,Z 623.616,A -85,B 0,C 180,E1 -6516.356,E2 -6516.356} C_VEL
LIN {X 0,Y 488.699,Z 623.613,A -85,B 0,C 180,E1 -6519.255,E2 -6519.255} C_VEL
LIN {X 0,Y 488.705,Z 623.612,A -85,B 0,C 180,E1 -6521.6,E2 -6521.6} C_VEL
LIN {X 0,Y 488.71,Z 623.612,A -85,B 0,C 180,E1 -6524.802,E2 -6524.802} C_VEL
LIN {X 0,Y 488.69,Z 623.615,A -85,B 0,C 180,E1 -6527.475,E2 -6527.475} C_VEL
LIN {X 0,Y 488.731,Z 623.61,A -85,B 0,C 180,E1 -6529.677,E2 -6529.677} C_VEL
LIN {X 0,Y 488.757,Z 623.72,A -85,B 0,C 180,E1 -6531.479,E2 -6531.479} C_VEL
LIN {X 0,Y 489.542,Z 628.793,A -85,B 0,C 180,E1 -6533.942,E2 -6533.942} C_VEL
LIN {X 0,Y 489.48,Z 634.152,A -85,B 0,C 180,E1 -6536.384,E2 -6536.384} C_VEL
LIN {X 0,Y 489.178,Z 642.001,A -85,B 0,C 180,E1 -6539.812,E2 -6539.812} C_VEL
LIN {X 0,Y 488.9,Z 649.663,A -85,B 0,C 180,E1 -6543.032,E2 -6543.032} C_VEL
LIN {X 0,Y 488.673,Z 657.542,A -85,B 0,C 180,E1 -6546.254,E2 -6546.254} C_VEL
LIN {X 0,Y 488.521,Z 665.059,A -85,B 0,C 180,E1 -6549.246,E2 -6549.246} C_VEL
LIN {X 0,Y 488.322,Z 673.202,A -85,B 0,C 180,E1 -6552.409,E2 -6552.409} C_VEL
LIN {X 0,Y 488.208,Z 680.715,A -85,B 0,C 180,E1 -6555.289,E2 -6555.289} C_VEL
LIN {X 0,Y 490.352,Z 693.9,A -85,B 0,C 180,E1 -6555.686,E2 -6555.686} C_VEL
LIN {X 0,Y 490.752,Z 698.482,A -85,B 0,C 180,E1 -6555.857,E2 -6555.857} C_VEL
LIN {X 0,Y 490.401,Z 710.562,A -85,B 0,C 180,E1 -6556.375,E2 -6556.375} C_VEL
LIN {X 0,Y 490.006,Z 722.132,A -85,B 0,C 180,E1 -6557.039,E2 -6557.039} C_VEL
LIN {X 0,Y 489.635,Z 733.639,A -85,B 0,C 180,E1 -6557.883,E2 -6557.883} C_VEL
LIN {X 0,Y 489.225,Z 743.866,A -85,B 0,C 180,E1 -6558.818,E2 -6558.818} C_VEL
LIN {X 0,Y 488.866,Z 753.064,A -85,B 0,C 180,E1 -6559.857,E2 -6559.857} C_VEL
LIN {X 0,Y 488.507,Z 762.023,A -85,B 0,C 180,E1 -6561.104,E2 -6561.104} C_VEL
LIN {X 0,Y 488.246,Z 769.236,A -85,B 0,C 180,E1 -6562.349,E2 -6562.349} C_VEL
LIN {X 0,Y 488.06,Z 775.617,A -85,B 0,C 180,E1 -6563.753,E2 -6563.753} C_VEL
LIN {X 0,Y 487.971,Z 780.148,A -85,B 0,C 180,E1 -6565.043,E2 -6565.043} C_VEL
LIN {X 0,Y 487.942,Z 782.447,A -85,B 0,C 180,E1 -6565.871,E2 -6565.871} C_VEL
LIN {X 0,Y 487.966,Z 784.312,A -85,B 0,C 180,E1 -6566.698,E2 -6566.698} C_VEL
LIN {X 0,Y 487.888,Z 786.704,A -85,B 0,C 180,E1 -6568.349,E2 -6568.349} C_VEL
LIN {X 0,Y 487.819,Z 787.524,A -85,B 0,C 180,E1 -6570,E2 -6570} C_VEL
LIN {X 0,Y 487.889,Z 786.698,A -85,B 0,C 180,E1 -6571.651,E2 -6571.651} C_VEL
LIN {X 0,Y 487.966,Z 784.299,A -85,B 0,C 180,E1 -6573.303,E2 -6573.303} C_VEL
LIN {X 0,Y 487.937,Z 781.351,A -85,B 0,C 180,E1 -6574.544,E2 -6574.544} C_VEL
LIN {X 0,Y 488.089,Z 777.367,A -85,B 0,C 180,E1 -6575.785,E2 -6575.785} C_VEL
LIN {X 0,Y 488.183,Z 771.233,A -85,B 0,C 180,E1 -6577.237,E2 -6577.237} C_VEL
LIN {X 0,Y 488.407,Z 764.533,A -85,B 0,C 180,E1 -6578.482,E2 -6578.482} C_VEL
LIN {X 0,Y 488.718,Z 756.217,A -85,B 0,C 180,E1 -6579.728,E2 -6579.728} C_VEL
LIN {X 0,Y 489.033,Z 747.689,A -85,B 0,C 180,E1 -6580.768,E2 -6580.768} C_VEL
LIN {X 0,Y 489.523,Z 737.16,A -85,B 0,C 180,E1 -6581.805,E2 -6581.805} C_VEL
LIN {X 0,Y 489.85,Z 726.194,A -85,B 0,C 180,E1 -6582.679,E2 -6582.679} C_VEL
LIN {X 0,Y 490.214,Z 715.326,A -85,B 0,C 180,E1 -6583.367,E2 -6583.367} C_VEL
LIN {X 0,Y 490.606,Z 703.588,A -85,B 0,C 180,E1 -6583.936,E2 -6583.936} C_VEL
LIN {X 0,Y 490.613,Z 695.617,A -85,B 0,C 180,E1 -6584.24,E2 -6584.24} C_VEL
LIN {X 0,Y 488.395,Z 682.263,A -85,B 0,C 180,E1 -6584.672,E2 -6584.672} C_VEL
LIN {X 0,Y 488.183,Z 680.468,A -85,B 0,C 180,E1 -6584.752,E2 -6584.752} C_VEL
LIN {X 0,Y 488.299,Z 672.989,A -85,B 0,C 180,E1 -6587.593,E2 -6587.593} C_VEL
LIN {X 0,Y 488.512,Z 664.777,A -85,B 0,C 180,E1 -6590.751,E2 -6590.751} C_VEL
LIN {X 0,Y 488.624,Z 657.173,A -85,B 0,C 180,E1 -6593.749,E2 -6593.749} C_VEL
LIN {X 0,Y 488.801,Z 650.481,A -85,B 0,C 180,E1 -6596.47,E2 -6596.47} C_VEL
LIN {X 0,Y 489.053,Z 643.871,A -85,B 0,C 180,E1 -6599.249,E2 -6599.249} C_VEL
LIN {X 0,Y 489.348,Z 636.234,A -85,B 0,C 180,E1 -6602.587,E2 -6602.587} C_VEL
LIN {X 0,Y 489.576,Z 629.808,A -85,B 0,C 180,E1 -6605.548,E2 -6605.548} C_VEL
LIN {X 0,Y 489.048,Z 625.347,A -85,B 0,C 180,E1 -6607.778,E2 -6607.778} C_VEL
LIN {X 0,Y 488.743,Z 623.605,A -85,B 0,C 180,E1 -6608.72,E2 -6608.72} C_VEL
LIN {X 0,Y 488.726,Z 623.611,A -85,B 0,C 180,E1 -6611.602,E2 -6611.602} C_VEL
LIN {X 0,Y 488.714,Z 623.611,A -85,B 0,C 180,E1 -6614.801,E2 -6614.801} C_VEL
LIN {X 0,Y 488.693,Z 623.615,A -85,B 0,C 180,E1 -6617.474,E2 -6617.474} C_VEL
LIN {X 0,Y 488.735,Z 623.61,A -85,B 0,C 180,E1 -6619.677,E2 -6619.677} C_VEL
LIN {X 0,Y 488.682,Z 623.615,A -85,B 0,C 180,E1 -6622.841,E2 -6622.841} C_VEL
LIN {X 0,Y 488.735,Z 623.607,A -85,B 0,C 180,E1 -6625.887,E2 -6625.887} C_VEL
LIN {X 0,Y 488.694,Z 623.613,A -85,B 0,C 180,E1 -6628.82,E2 -6628.82} C_VEL
LIN {X 0,Y 488.746,Z 623.607,A -85,B 0,C 180,E1 -6631.671,E2 -6631.671} C_VEL
LIN {X 0,Y 488.749,Z 623.607,A -85,B 0,C 180,E1 -6634.444,E2 -6634.444} C_VEL
LIN {X 0,Y 488.726,Z 623.609,A -85,B 0,C 180,E1 -6637.153,E2 -6637.153} C_VEL
LIN {X 0,Y 488.73,Z 623.609,A -85,B 0,C 180,E1 -6639.811,E2 -6639.811} C_VEL
LIN {X 0,Y 488.736,Z 623.609,A -85,B 0,C 180,E1 -6642.423,E2 -6642.423} C_VEL
LIN {X 0,Y 488.764,Z 623.604,A -85,B 0,C 180,E1 -6645,E2 -6645} C_VEL
LIN {X 0,Y 488.807,Z 623.6,A -85,B 0,C 180,E1 -6648.388,E2 -6648.388} C_VEL
LIN {X 0,Y 488.82,Z 623.598,A -85,B 0,C 180,E1 -6651.734,E2 -6651.734} C_VEL
LIN {X 0,Y 488.857,Z 623.592,A -85,B 0,C 180,E1 -6654.224,E2 -6654.224} C_VEL
LIN {X 0,Y 488.962,Z 623.58,A -85,B 0,C 180,E1 -6657.529,E2 -6657.529} C_VEL
LIN {X 0,Y 488.957,Z 623.583,A -85,B 0,C 180,E1 -6660.824,E2 -6660.824} C_VEL
LIN {X 0,Y 488.963,Z 623.581,A -85,B 0,C 180,E1 -6662.471,E2 -6662.471} C_VEL
LIN {X 0,Y 488.858,Z 623.594,A -85,B 0,C 180,E1 -6665.776,E2 -6665.776} C_VEL
LIN {X 0,Y 488.806,Z 623.6,A -85,B 0,C 180,E1 -6668.267,E2 -6668.267} C_VEL
LIN {X 0,Y 488.737,Z 623.609,A -85,B 0,C 180,E1 -6669.101,E2 -6669.101} C_VEL
LIN {X 0,Y 488.706,Z 624.102,A -85,B 0,C 180,E1 -6669.937,E2 -6669.937} C_VEL
LIN {X 0,Y 488.612,Z 627.636,A -85,B 0,C 180,E1 -6672.46,E2 -6672.46} C_VEL
LIN {X 0,Y 488.466,Z 632.532,A -85,B 0,C 180,E1 -6675.865,E2 -6675.865} C_VEL
LIN {X 0,Y 488.359,Z 636.313,A -85,B 0,C 180,E1 -6678.458,E2 -6678.458} C_VEL
LIN {X 0,Y 488.262,Z 640.277,A -85,B 0,C 180,E1 -6681.091,E2 -6681.091} C_VEL
LIN {X 0,Y 488.13,Z 644.364,A -85,B 0,C 180,E1 -6683.775,E2 -6683.775} C_VEL
LIN {X 0,Y 488.098,Z 649,A -85,B 0,C 180,E1 -6686.783,E2 -6686.783} C_VEL
LIN {X 0,Y 487.99,Z 652.962,A -85,B 0,C 180,E1 -6689.319,E2 -6689.319} C_VEL
LIN {X 0,Y 487.964,Z 654.612,A -85,B 0,C 180,E1 -6690.361,E2 -6690.361} C_VEL
LIN {X 0,Y 490.432,Z 667.182,A -85,B 0,C 180,E1 -6690.788,E2 -6690.788} C_VEL
LIN {X 0,Y 490.806,Z 670.363,A -85,B 0,C 180,E1 -6690.911,E2 -6690.911} C_VEL
LIN {X 0,Y 490.484,Z 683.167,A -85,B 0,C 180,E1 -6691.474,E2 -6691.474} C_VEL
